LIN {X 0,Y 301.636,Z 553.215,A -85,B 0,C 180,E1 -16563.673,E2 -16563.673} C_VEL
LIN {X 0,Y 304.544,Z 543.643,A -85,B 0,C 180,E1 -16565.661,E2 -16565.661} C_VEL
LIN {X 0,Y 307.62,Z 532.508,A -85,B 0,C 180,E1 -16567.548,E2 -16567.548} C_VEL
LIN {X 0,Y 310.787,Z 520.04,A -85,B 0,C 180,E1 -16569.269,E2 -16569.269} C_VEL
LIN {X 0,Y 312.325,Z 513.549,A -85,B 0,C 180,E1 -16570.029,E2 -16570.029} C_VEL
LIN {X 0,Y 311.304,Z 507.375,A -85,B 0,C 180,E1 -16571.095,E2 -16571.095} C_VEL
LIN {X 0,Y 308.956,Z 499.343,A -85,B 0,C 180,E1 -16572.599,E2 -16572.599} C_VEL
LIN {X 0,Y 305.518,Z 490.599,A -85,B 0,C 180,E1 -16574.386,E2 -16574.386} C_VEL
LIN {X 0,Y 301.49,Z 482.379,A -85,B 0,C 180,E1 -16576.244,E2 -16576.244} C_VEL
LIN {X 0,Y 299.043,Z 478.041,A -85,B 0,C 180,E1 -16577.361,E2 -16577.361} C_VEL
LIN {X 0,Y 296.682,Z 474.656,A -85,B 0,C 180,E1 -16578.369,E2 -16578.369} C_VEL
LIN {X 0,Y 295.976,Z 473.129,A -85,B 0,C 180,E1 -16578.748,E2 -16578.748} C_VEL
LIN {X 0,Y 293.748,Z 470.591,A -85,B 0,C 180,E1 -16579.696,E2 -16579.696} C_VEL
LIN {X 0,Y 292.906,Z 468.275,A -85,B 0,C 180,E1 -16580.21,E2 -16580.21} C_VEL
LIN {X 0,Y 293.027,Z 467.949,A -85,B 0,C 180,E1 -16584.303,E2 -16584.303} C_VEL
LIN {X 0,Y 293.139,Z 468.076,A -85,B 0,C 180,E1 -16587.494,E2 -16587.494} C_VEL
LIN {X 0,Y 293.233,Z 468.47,A -85,B 0,C 180,E1 -16590.367,E2 -16590.367} C_VEL
LIN {X 0,Y 293.482,Z 469.78,A -85,B 0,C 180,E1 -16595.08,E2 -16595.08} C_VEL
LIN {X 0,Y 293.714,Z 471.269,A -85,B 0,C 180,E1 -16598.472,E2 -16598.472} C_VEL
LIN {X 0,Y 294.132,Z 473.425,A -85,B 0,C 180,E1 -16602.209,E2 -16602.209} C_VEL
LIN {X 0,Y 294.599,Z 476.404,A -85,B 0,C 180,E1 -16606.226,E2 -16606.226} C_VEL
LIN {X 0,Y 294.714,Z 478.064,A -85,B 0,C 180,E1 -16608.11,E2 -16608.11} C_VEL
LIN {X 0,Y 294.685,Z 479.821,A -85,B 0,C 180,E1 -16609.916,E2 -16609.916} C_VEL
LIN {X 0,Y 294.321,Z 482.209,A -85,B 0,C 180,E1 -16612.14,E2 -16612.14} C_VEL
LIN {X 0,Y 295.331,Z 485.828,A -85,B 0,C 180,E1 -16612.78,E2 -16612.78} C_VEL
LIN {X 0,Y 296.885,Z 488.688,A -85,B 0,C 180,E1 -16613.453,E2 -16613.453} C_VEL
LIN {X 0,Y 298.233,Z 492.616,A -85,B 0,C 180,E1 -16614.157,E2 -16614.157} C_VEL
LIN {X 0,Y 299.091,Z 494.768,A -85,B 0,C 180,E1 -16614.576,E2 -16614.576} C_VEL
LIN {X 0,Y 302.369,Z 504.747,A -85,B 0,C 180,E1 -16616.289,E2 -16616.289} C_VEL
LIN {X 0,Y 305.21,Z 516.489,A -85,B 0,C 180,E1 -16618.121,E2 -16618.121} C_VEL
LIN {X 0,Y 306.937,Z 528.969,A -85,B 0,C 180,E1 -16619.932,E2 -16619.932} C_VEL
LIN {X 0,Y 307.426,Z 538.705,A -85,B 0,C 180,E1 -16621.31,E2 -16621.31} C_VEL
LIN {X 0,Y 306.788,Z 549.97,A -85,B 0,C 180,E1 -16622.916,E2 -16622.916} C_VEL
LIN {X 0,Y 305.504,Z 555.839,A -85,B 0,C 180,E1 -16623.715,E2 -16623.715} C_VEL
LIN {X 0,Y 302.625,Z 566.34,A -85,B 0,C 180,E1 -16625.291,E2 -16625.291} C_VEL
LIN {X 0,Y 299.636,Z 576.972,A -85,B 0,C 180,E1 -16627.232,E2 -16627.232} C_VEL
LIN {X 0,Y 296.657,Z 587.405,A -85,B 0,C 180,E1 -16629.547,E2 -16629.547} C_VEL
LIN {X 0,Y 294.253,Z 596.056,A -85,B 0,C 180,E1 -16631.911,E2 -16631.911} C_VEL
LIN {X 0,Y 292.244,Z 604.121,A -85,B 0,C 180,E1 -16634.661,E2 -16634.661} C_VEL
LIN {X 0,Y 290.802,Z 610.467,A -85,B 0,C 180,E1 -16637.437,E2 -16637.437} C_VEL
LIN {X 0,Y 289.949,Z 615.257,A -85,B 0,C 180,E1 -16640.231,E2 -16640.231} C_VEL
LIN {X 0,Y 289.566,Z 618.621,A -85,B 0,C 180,E1 -16643.03,E2 -16643.03} C_VEL
LIN {X 0,Y 289.558,Z 620.61,A -85,B 0,C 180,E1 -16645.824,E2 -16645.824} C_VEL
LIN {X 0,Y 289.675,Z 621.212,A -85,B 0,C 180,E1 -16648.61,E2 -16648.61} C_VEL
LIN {X 0,Y 289.873,Z 620.996,A -85,B 0,C 180,E1 -16650,E2 -16650} C_VEL
LIN {X 0,Y 289.631,Z 619.447,A -85,B 0,C 180,E1 -16652.782,E2 -16652.782} C_VEL
LIN {X 0,Y 289.672,Z 618.137,A -85,B 0,C 180,E1 -16654.174,E2 -16654.174} C_VEL
LIN {X 0,Y 289.71,Z 615.903,A -85,B 0,C 180,E1 -16655.954,E2 -16655.954} C_VEL
LIN {X 0,Y 289.811,Z 611.833,A -85,B 0,C 180,E1 -16658.366,E2 -16658.366} C_VEL
LIN {X 0,Y 290.092,Z 607.241,A -85,B 0,C 180,E1 -16660.469,E2 -16660.469} C_VEL
LIN {X 0,Y 290.817,Z 600.58,A -85,B 0,C 180,E1 -16662.917,E2 -16662.917} C_VEL
LIN {X 0,Y 291.753,Z 592.22,A -85,B 0,C 180,E1 -16665.365,E2 -16665.365} C_VEL
LIN {X 0,Y 293.093,Z 583.538,A -85,B 0,C 180,E1 -16667.441,E2 -16667.441} C_VEL
LIN {X 0,Y 294.652,Z 573.049,A -85,B 0,C 180,E1 -16669.507,E2 -16669.507} C_VEL
LIN {X 0,Y 296.588,Z 561.479,A -85,B 0,C 180,E1 -16671.366,E2 -16671.366} C_VEL
LIN {X 0,Y 298.446,Z 548.652,A -85,B 0,C 180,E1 -16673.047,E2 -16673.047} C_VEL
LIN {X 0,Y 298.999,Z 544.142,A -85,B 0,C 180,E1 -16673.552,E2 -16673.552} C_VEL
LIN {X 0,Y 297.569,Z 530.241,A -85,B 0,C 180,E1 -16675.065,E2 -16675.065} C_VEL
LIN {X 0,Y 295.6,Z 515.743,A -85,B 0,C 180,E1 -16676.36,E2 -16676.36} C_VEL
LIN {X 0,Y 293.096,Z 500.193,A -85,B 0,C 180,E1 -16677.476,E2 -16677.476} C_VEL
LIN {X 0,Y 291.412,Z 490.807,A -85,B 0,C 180,E1 -16678.051,E2 -16678.051} C_VEL
LIN {X 0,Y 292.233,Z 484.923,A -85,B 0,C 180,E1 -16681.943,E2 -16681.943} C_VEL
LIN {X 0,Y 293.22,Z 478.9,A -85,B 0,C 180,E1 -16686.02,E2 -16686.02} C_VEL
LIN {X 0,Y 293.911,Z 474.253,A -85,B 0,C 180,E1 -16689.252,E2 -16689.252} C_VEL
LIN {X 0,Y 293.611,Z 470.39,A -85,B 0,C 180,E1 -16692.096,E2 -16692.096} C_VEL
LIN {X 0,Y 292.747,Z 465.551,A -85,B 0,C 180,E1 -16695.877,E2 -16695.877} C_VEL
LIN {X 0,Y 291.997,Z 461.184,A -85,B 0,C 180,E1 -16699.469,E2 -16699.469} C_VEL
LIN {X 0,Y 291.434,Z 457.811,A -85,B 0,C 180,E1 -16702.434,E2 -16702.434} C_VEL
LIN {X 0,Y 291.342,Z 457.816,A -85,B 0,C 180,E1 -16706.301,E2 -16706.301} C_VEL
LIN {X 0,Y 291.384,Z 457.812,A -85,B 0,C 180,E1 -16710.259,E2 -16710.259} C_VEL
LIN {X 0,Y 291.412,Z 457.807,A -85,B 0,C 180,E1 -16714.272,E2 -16714.272} C_VEL
LIN {X 0,Y 291.377,Z 457.814,A -85,B 0,C 180,E1 -16717.299,E2 -16717.299} C_VEL
LIN {X 0,Y 291.454,Z 457.803,A -85,B 0,C 180,E1 -16720.27,E2 -16720.27} C_VEL
LIN {X 0,Y 291.551,Z 457.793,A -85,B 0,C 180,E1 -16724.624,E2 -16724.624} C_VEL
LIN {X 0,Y 291.532,Z 457.797,A -85,B 0,C 180,E1 -16728.881,E2 -16728.881} C_VEL
LIN {X 0,Y 291.704,Z 457.771,A -85,B 0,C 180,E1 -16731.689,E2 -16731.689} C_VEL
LIN {X 0,Y 291.627,Z 457.783,A -85,B 0,C 180,E1 -16734.469,E2 -16734.469} C_VEL
LIN {X 0,Y 291.886,Z 457.754,A -85,B 0,C 180,E1 -16738.621,E2 -16738.621} C_VEL
LIN {X 0,Y 291.888,Z 457.748,A -85,B 0,C 180,E1 -16741.38,E2 -16741.38} C_VEL
LIN {X 0,Y 291.744,Z 457.768,A -85,B 0,C 180,E1 -16746.918,E2 -16746.918} C_VEL
LIN {X 0,Y 291.625,Z 457.781,A -85,B 0,C 180,E1 -16749.712,E2 -16749.712} C_VEL
LIN {X 0,Y 291.517,Z 457.796,A -85,B 0,C 180,E1 -16753.951,E2 -16753.951} C_VEL
LIN {X 0,Y 291.483,Z 457.8,A -85,B 0,C 180,E1 -16756.818,E2 -16756.818} C_VEL
LIN {X 0,Y 291.447,Z 457.804,A -85,B 0,C 180,E1 -16759.875,E2 -16759.875} C_VEL
LIN {X 0,Y 291.397,Z 457.814,A -85,B 0,C 180,E1 -16764.206,E2 -16764.206} C_VEL
LIN {X 0,Y 291.419,Z 457.806,A -85,B 0,C 180,E1 -16767.272,E2 -16767.272} C_VEL
LIN {X 0,Y 291.334,Z 457.82,A -85,B 0,C 180,E1 -16770.438,E2 -16770.438} C_VEL
LIN {X 0,Y 291.342,Z 457.818,A -85,B 0,C 180,E1 -16773.699,E2 -16773.699} C_VEL
LIN {X 0,Y 291.379,Z 457.811,A -85,B 0,C 180,E1 -16777.256,E2 -16777.256} C_VEL
LIN {X 0,Y 291.332,Z 457.819,A -85,B 0,C 180,E1 -16780.643,E2 -16780.643} C_VEL
LIN {X 0,Y 291.289,Z 457.824,A -85,B 0,C 180,E1 -16784.403,E2 -16784.403} C_VEL
LIN {X 0,Y 291.355,Z 457.816,A -85,B 0,C 180,E1 -16788.399,E2 -16788.399} C_VEL
LIN {X 0,Y 291.38,Z 457.812,A -85,B 0,C 180,E1 -16791.163,E2 -16791.163} C_VEL
LIN {X 0,Y 291.386,Z 457.81,A -85,B 0,C 180,E1 -16794.63,E2 -16794.63} C_VEL
LIN {X 0,Y 291.374,Z 457.816,A -85,B 0,C 180,E1 -16797.952,E2 -16797.952} C_VEL
LIN {X 0,Y 291.391,Z 457.811,A -85,B 0,C 180,E1 -16801.16,E2 -16801.16} C_VEL
LIN {X 0,Y 291.423,Z 457.807,A -85,B 0,C 180,E1 -16804.273,E2 -16804.273} C_VEL
LIN {X 0,Y 291.384,Z 457.813,A -85,B 0,C 180,E1 -16807.3,E2 -16807.3} C_VEL
LIN {X 0,Y 291.461,Z 457.802,A -85,B 0,C 180,E1 -16810.271,E2 -16810.271} C_VEL
LIN {X 0,Y 291.558,Z 457.789,A -85,B 0,C 180,E1 -16814.624,E2 -16814.624} C_VEL
LIN {X 0,Y 291.539,Z 457.792,A -85,B 0,C 180,E1 -16818.881,E2 -16818.881} C_VEL
LIN {X 0,Y 291.658,Z 457.78,A -85,B 0,C 180,E1 -16821.687,E2 -16821.687} C_VEL
LIN {X 0,Y 291.615,Z 457.782,A -85,B 0,C 180,E1 -16824.468,E2 -16824.468} C_VEL
LIN {X 0,Y 291.892,Z 457.747,A -85,B 0,C 180,E1 -16828.62,E2 -16828.62} C_VEL
LIN {X 0,Y 291.892,Z 457.752,A -85,B 0,C 180,E1 -16831.38,E2 -16831.38} C_VEL
LIN {X 0,Y 291.738,Z 457.769,A -85,B 0,C 180,E1 -16836.918,E2 -16836.918} C_VEL
LIN {X 0,Y 291.578,Z 457.787,A -85,B 0,C 180,E1 -16839.713,E2 -16839.713} C_VEL
LIN {X 0,Y 291.525,Z 457.794,A -85,B 0,C 180,E1 -16843.95,E2 -16843.95} C_VEL
LIN {X 0,Y 291.49,Z 457.8,A -85,B 0,C 180,E1 -16846.817,E2 -16846.817} C_VEL
LIN {X 0,Y 291.453,Z 457.803,A -85,B 0,C 180,E1 -16849.874,E2 -16849.874} C_VEL
LIN {X 0,Y 291.402,Z 457.809,A -85,B 0,C 180,E1 -16854.205,E2 -16854.205} C_VEL
LIN {X 0,Y 291.424,Z 457.81,A -85,B 0,C 180,E1 -16857.271,E2 -16857.271} C_VEL
LIN {X 0,Y 291.336,Z 457.819,A -85,B 0,C 180,E1 -16860.436,E2 -16860.436} C_VEL
LIN {X 0,Y 291.243,Z 457.829,A -85,B 0,C 180,E1 -16863.711,E2 -16863.711} C_VEL
LIN {X 0,Y 290.986,Z 457.864,A -85,B 0,C 180,E1 -16867.152,E2 -16867.152} C_VEL
LIN {X 0,Y 290.57,Z 457.917,A -85,B 0,C 180,E1 -16870.771,E2 -16870.771} C_VEL
LIN {X 0,Y 290.267,Z 458.188,A -85,B 0,C 180,E1 -16873.417,E2 -16873.417} C_VEL
LIN {X 0,Y 290.253,Z 458.716,A -85,B 0,C 180,E1 -16874.108,E2 -16874.108} C_VEL
LIN {X 0,Y 295.016,Z 475.364,A -85,B 0,C 180,E1 -16875.334,E2 -16875.334} C_VEL
LIN {X 0,Y 298.444,Z 488.673,A -85,B 0,C 180,E1 -16876.532,E2 -16876.532} C_VEL
LIN {X 0,Y 300.997,Z 500.048,A -85,B 0,C 180,E1 -16877.735,E2 -16877.735} C_VEL
LIN {X 0,Y 299.772,Z 511.987,A -85,B 0,C 180,E1 -16878.97,E2 -16878.97} C_VEL
LIN {X 0,Y 298.086,Z 523.963,A -85,B 0,C 180,E1 -16880.462,E2 -16880.462} C_VEL
LIN {X 0,Y 296.452,Z 535.158,A -85,B 0,C 180,E1 -16882.162,E2 -16882.162} C_VEL
LIN {X 0,Y 294.809,Z 545.907,A -85,B 0,C 180,E1 -16884.146,E2 -16884.146} C_VEL
LIN {X 0,Y 293.434,Z 554.954,A -85,B 0,C 180,E1 -16886.161,E2 -16886.161} C_VEL
LIN {X 0,Y 292.141,Z 563.427,A -85,B 0,C 180,E1 -16888.45,E2 -16888.45} C_VEL
LIN {X 0,Y 291.228,Z 570.208,A -85,B 0,C 180,E1 -16890.689,E2 -16890.689} C_VEL
LIN {X 0,Y 290.465,Z 576.263,A -85,B 0,C 180,E1 -16893.175,E2 -16893.175} C_VEL
LIN {X 0,Y 289.946,Z 580.967,A -85,B 0,C 180,E1 -16895.665,E2 -16895.665} C_VEL
LIN {X 0,Y 289.734,Z 583.225,A -85,B 0,C 180,E1 -16897.181,E2 -16897.181} C_VEL
LIN {X 0,Y 289.45,Z 586.399,A -85,B 0,C 180,E1 -16900.127,E2 -16900.127} C_VEL
LIN {X 0,Y 289.497,Z 587.383,A -85,B 0,C 180,E1 -16901.603,E2 -16901.603} C_VEL
LIN {X 0,Y 289.655,Z 588.2,A -85,B 0,C 180,E1 -16904.52,E2 -16904.52} C_VEL
LIN {X 0,Y 290.106,Z 587.576,A -85,B 0,C 180,E1 -16907.406,E2 -16907.406} C_VEL
LIN {X 0,Y 290.896,Z 585.558,A -85,B 0,C 180,E1 -16910.263,E2 -16910.263} C_VEL
LIN {X 0,Y 292.112,Z 582.127,A -85,B 0,C 180,E1 -16913.09,E2 -16913.09} C_VEL
LIN {X 0,Y 293.789,Z 577.212,A -85,B 0,C 180,E1 -16915.884,E2 -16915.884} C_VEL
LIN {X 0,Y 296.006,Z 570.651,A -85,B 0,C 180,E1 -16918.639,E2 -16918.639} C_VEL
LIN {X 0,Y 296.133,Z 570.261,A -85,B 0,C 180,E1 -16918.78,E2 -16918.78} C_VEL
LIN {X 0,Y 296.44,Z 567.593,A -85,B 0,C 180,E1 -16919.797,E2 -16919.797} C_VEL
LIN {X 0,Y 295.401,Z 563.24,A -85,B 0,C 180,E1 -16921.513,E2 -16921.513} C_VEL
LIN {X 0,Y 294.562,Z 558.444,A -85,B 0,C 180,E1 -16923.185,E2 -16923.185} C_VEL
LIN {X 0,Y 295.151,Z 555.046,A -85,B 0,C 180,E1 -16924.112,E2 -16924.112} C_VEL
LIN {X 0,Y 298.125,Z 545.908,A -85,B 0,C 180,E1 -16926.105,E2 -16926.105} C_VEL
LIN {X 0,Y 301.368,Z 535.215,A -85,B 0,C 180,E1 -16928.043,E2 -16928.043} C_VEL
LIN {X 0,Y 304.666,Z 523.197,A -85,B 0,C 180,E1 -16929.795,E2 -16929.795} C_VEL
LIN {X 0,Y 306.496,Z 515.55,A -85,B 0,C 180,E1 -16930.745,E2 -16930.745} C_VEL
LIN {X 0,Y 305.179,Z 508.082,A -85,B 0,C 180,E1 -16932.161,E2 -16932.161} C_VEL
LIN {X 0,Y 302.061,Z 498.218,A -85,B 0,C 180,E1 -16934.202,E2 -16934.202} C_VEL
LIN {X 0,Y 297.217,Z 487.393,A -85,B 0,C 180,E1 -16936.79,E2 -16936.79} C_VEL
LIN {X 0,Y 294.604,Z 482.84,A -85,B 0,C 180,E1 -16938.067,E2 -16938.067} C_VEL
LIN {X 0,Y 291.609,Z 478.107,A -85,B 0,C 180,E1 -16939.582,E2 -16939.582} C_VEL
LIN {X 0,Y 289.874,Z 475.066,A -85,B 0,C 180,E1 -16940.55,E2 -16940.55} C_VEL
LIN {X 0,Y 289.424,Z 474.387,A -85,B 0,C 180,E1 -16940.797,E2 -16940.797} C_VEL
LIN {X 0,Y 287.052,Z 472.053,A -85,B 0,C 180,E1 -16941.97,E2 -16941.97} C_VEL
LIN {X 0,Y 286.042,Z 469.515,A -85,B 0,C 180,E1 -16942.728,E2 -16942.728} C_VEL
LIN {X 0,Y 286.142,Z 469.511,A -85,B 0,C 180,E1 -16946.238,E2 -16946.238} C_VEL
LIN {X 0,Y 286.237,Z 469.877,A -85,B 0,C 180,E1 -16949.41,E2 -16949.41} C_VEL
LIN {X 0,Y 286.413,Z 470.819,A -85,B 0,C 180,E1 -16953.459,E2 -16953.459} C_VEL
LIN {X 0,Y 286.746,Z 472.49,A -85,B 0,C 180,E1 -16957.787,E2 -16957.787} C_VEL
LIN {X 0,Y 287.094,Z 474.43,A -85,B 0,C 180,E1 -16961.373,E2 -16961.373} C_VEL
LIN {X 0,Y 287.528,Z 477.024,A -85,B 0,C 180,E1 -16965.141,E2 -16965.141} C_VEL
LIN {X 0,Y 287.714,Z 478.619,A -85,B 0,C 180,E1 -16967.122,E2 -16967.122} C_VEL
LIN {X 0,Y 287.741,Z 481.304,A -85,B 0,C 180,E1 -16969.887,E2 -16969.887} C_VEL
LIN {X 0,Y 288.623,Z 484.501,A -85,B 0,C 180,E1 -16970.542,E2 -16970.542} C_VEL
LIN {X 0,Y 290.726,Z 488.229,A -85,B 0,C 180,E1 -16971.611,E2 -16971.611} C_VEL
LIN {X 0,Y 292.274,Z 492.398,A -85,B 0,C 180,E1 -16972.515,E2 -16972.515} C_VEL
LIN {X 0,Y 293.032,Z 494.501,A -85,B 0,C 180,E1 -16972.961,E2 -16972.961} C_VEL
LIN {X 0,Y 295.012,Z 500.212,A -85,B 0,C 180,E1 -16974.093,E2 -16974.093} C_VEL
LIN {X 0,Y 297.161,Z 507.283,A -85,B 0,C 180,E1 -16975.417,E2 -16975.417} C_VEL
LIN {X 0,Y 299.741,Z 518.981,A -85,B 0,C 180,E1 -16977.366,E2 -16977.366} C_VEL
LIN {X 0,Y 301.182,Z 530.305,A -85,B 0,C 180,E1 -16979.112,E2 -16979.112} C_VEL
LIN {X 0,Y 301.471,Z 540.725,A -85,B 0,C 180,E1 -16980.689,E2 -16980.689} C_VEL
LIN {X 0,Y 300.65,Z 551.565,A -85,B 0,C 180,E1 -16982.316,E2 -16982.316} C_VEL
LIN {X 0,Y 298.932,Z 558.293,A -85,B 0,C 180,E1 -16983.28,E2 -16983.28} C_VEL
LIN {X 0,Y 295.705,Z 569.214,A -85,B 0,C 180,E1 -16985.048,E2 -16985.048} C_VEL
LIN {X 0,Y 292.682,Z 579.34,A -85,B 0,C 180,E1 -16987.033,E2 -16987.033} C_VEL
LIN {X 0,Y 289.615,Z 589.228,A -85,B 0,C 180,E1 -16989.399,E2 -16989.399} C_VEL
LIN {X 0,Y 287.19,Z 597.442,A -85,B 0,C 180,E1 -16991.82,E2 -16991.82} C_VEL
LIN {X 0,Y 285.366,Z 604.23,A -85,B 0,C 180,E1 -16994.282,E2 -16994.282} C_VEL
LIN {X 0,Y 283.848,Z 610.397,A -85,B 0,C 180,E1 -16997.124,E2 -16997.124} C_VEL
LIN {X 0,Y 282.886,Z 615.084,A -85,B 0,C 180,E1 -16999.985,E2 -16999.985} C_VEL
LIN {X 0,Y 282.484,Z 618.345,A -85,B 0,C 180,E1 -17002.854,E2 -17002.854} C_VEL
LIN {X 0,Y 282.472,Z 620.237,A -85,B 0,C 180,E1 -17005.719,E2 -17005.719} C_VEL
LIN {X 0,Y 282.584,Z 620.751,A -85,B 0,C 180,E1 -17008.575,E2 -17008.575} C_VEL
LIN {X 0,Y 282.801,Z 620.49,A -85,B 0,C 180,E1 -17010,E2 -17010} C_VEL
LIN {X 0,Y 282.555,Z 618.847,A -85,B 0,C 180,E1 -17012.851,E2 -17012.851} C_VEL
LIN {X 0,Y 282.61,Z 617.487,A -85,B 0,C 180,E1 -17014.278,E2 -17014.278} C_VEL
LIN {X 0,Y 282.646,Z 615.367,A -85,B 0,C 180,E1 -17015.957,E2 -17015.957} C_VEL
LIN {X 0,Y 282.744,Z 610.982,A -85,B 0,C 180,E1 -17018.577,E2 -17018.577} C_VEL
LIN {X 0,Y 283.058,Z 606.337,A -85,B 0,C 180,E1 -17020.732,E2 -17020.732} C_VEL
LIN {X 0,Y 283.824,Z 599.54,A -85,B 0,C 180,E1 -17023.241,E2 -17023.241} C_VEL
LIN {X 0,Y 284.87,Z 591.046,A -85,B 0,C 180,E1 -17025.746,E2 -17025.746} C_VEL
LIN {X 0,Y 286.245,Z 582.229,A -85,B 0,C 180,E1 -17027.872,E2 -17027.872} C_VEL
LIN {X 0,Y 287.88,Z 571.595,A -85,B 0,C 180,E1 -17029.985,E2 -17029.985} C_VEL
LIN {X 0,Y 289.861,Z 559.834,A -85,B 0,C 180,E1 -17031.887,E2 -17031.887} C_VEL
LIN {X 0,Y 291.651,Z 547.852,A -85,B 0,C 180,E1 -17033.467,E2 -17033.467} C_VEL
LIN {X 0,Y 292.019,Z 544.439,A -85,B 0,C 180,E1 -17033.859,E2 -17033.859} C_VEL
LIN {X 0,Y 290.737,Z 531.607,A -85,B 0,C 180,E1 -17035.312,E2 -17035.312} C_VEL
LIN {X 0,Y 288.918,Z 517.699,A -85,B 0,C 180,E1 -17036.627,E2 -17036.627} C_VEL
LIN {X 0,Y 286.552,Z 502.648,A -85,B 0,C 180,E1 -17037.774,E2 -17037.774} C_VEL
LIN {X 0,Y 284.415,Z 490.492,A -85,B 0,C 180,E1 -17038.536,E2 -17038.536} C_VEL
LIN {X 0,Y 285.176,Z 485.419,A -85,B 0,C 180,E1 -17041.995,E2 -17041.995} C_VEL
LIN {X 0,Y 286.177,Z 479.481,A -85,B 0,C 180,E1 -17046.114,E2 -17046.114} C_VEL
LIN {X 0,Y 286.862,Z 474.662,A -85,B 0,C 180,E1 -17049.567,E2 -17049.567} C_VEL
LIN {X 0,Y 286.483,Z 470.667,A -85,B 0,C 180,E1 -17052.612,E2 -17052.612} C_VEL
LIN {X 0,Y 285.616,Z 465.894,A -85,B 0,C 180,E1 -17056.451,E2 -17056.451} C_VEL
LIN {X 0,Y 284.848,Z 461.598,A -85,B 0,C 180,E1 -17060.097,E2 -17060.097} C_VEL
LIN {X 0,Y 284.412,Z 458.685,A -85,B 0,C 180,E1 -17062.746,E2 -17062.746} C_VEL
LIN {X 0,Y 284.303,Z 458.698,A -85,B 0,C 180,E1 -17067.055,E2 -17067.055} C_VEL
LIN {X 0,Y 284.356,Z 458.688,A -85,B 0,C 180,E1 -17070.376,E2 -17070.376} C_VEL
LIN {X 0,Y 284.374,Z 458.684,A -85,B 0,C 180,E1 -17073.586,E2 -17073.586} C_VEL
LIN {X 0,Y 284.362,Z 458.688,A -85,B 0,C 180,E1 -17076.707,E2 -17076.707} C_VEL
LIN {X 0,Y 284.399,Z 458.683,A -85,B 0,C 180,E1 -17081.262,E2 -17081.262} C_VEL
LIN {X 0,Y 284.488,Z 458.671,A -85,B 0,C 180,E1 -17084.459,E2 -17084.459} C_VEL
LIN {X 0,Y 284.484,Z 458.674,A -85,B 0,C 180,E1 -17088.602,E2 -17088.602} C_VEL
LIN {X 0,Y 284.654,Z 458.649,A -85,B 0,C 180,E1 -17091.481,E2 -17091.481} C_VEL
LIN {X 0,Y 284.597,Z 458.658,A -85,B 0,C 180,E1 -17094.331,E2 -17094.331} C_VEL
LIN {X 0,Y 284.852,Z 458.63,A -85,B 0,C 180,E1 -17098.587,E2 -17098.587} C_VEL
LIN {X 0,Y 284.854,Z 458.623,A -85,B 0,C 180,E1 -17101.414,E2 -17101.414} C_VEL
LIN {X 0,Y 284.695,Z 458.645,A -85,B 0,C 180,E1 -17107.09,E2 -17107.09} C_VEL
LIN {X 0,Y 284.562,Z 458.661,A -85,B 0,C 180,E1 -17109.956,E2 -17109.956} C_VEL
LIN {X 0,Y 284.474,Z 458.676,A -85,B 0,C 180,E1 -17114.304,E2 -17114.304} C_VEL
LIN {X 0,Y 284.421,Z 458.678,A -85,B 0,C 180,E1 -17117.249,E2 -17117.249} C_VEL
LIN {X 0,Y 284.375,Z 458.687,A -85,B 0,C 180,E1 -17120.243,E2 -17120.243} C_VEL
LIN {X 0,Y 284.366,Z 458.687,A -85,B 0,C 180,E1 -17123.876,E2 -17123.876} C_VEL
LIN {X 0,Y 284.394,Z 458.681,A -85,B 0,C 180,E1 -17127.174,E2 -17127.174} C_VEL
LIN {X 0,Y 284.293,Z 458.694,A -85,B 0,C 180,E1 -17131.275,E2 -17131.275} C_VEL
LIN {X 0,Y 284.339,Z 458.689,A -85,B 0,C 180,E1 -17135.349,E2 -17135.349} C_VEL
LIN {X 0,Y 284.317,Z 458.696,A -85,B 0,C 180,E1 -17138.169,E2 -17138.169} C_VEL
LIN {X 0,Y 284.268,Z 458.702,A -85,B 0,C 180,E1 -17142.125,E2 -17142.125} C_VEL
LIN {X 0,Y 284.272,Z 458.7,A -85,B 0,C 180,E1 -17146.193,E2 -17146.193} C_VEL
LIN {X 0,Y 284.351,Z 458.692,A -85,B 0,C 180,E1 -17150.014,E2 -17150.014} C_VEL
LIN {X 0,Y 284.353,Z 458.689,A -85,B 0,C 180,E1 -17153.618,E2 -17153.618} C_VEL
LIN {X 0,Y 284.309,Z 458.693,A -85,B 0,C 180,E1 -17157.19,E2 -17157.19} C_VEL
LIN {X 0,Y 284.363,Z 458.686,A -85,B 0,C 180,E1 -17160.377,E2 -17160.377} C_VEL
LIN {X 0,Y 284.383,Z 458.686,A -85,B 0,C 180,E1 -17163.588,E2 -17163.588} C_VEL
LIN {X 0,Y 284.369,Z 458.685,A -85,B 0,C 180,E1 -17166.708,E2 -17166.708} C_VEL
LIN {X 0,Y 284.407,Z 458.682,A -85,B 0,C 180,E1 -17171.262,E2 -17171.262} C_VEL
LIN {X 0,Y 284.495,Z 458.669,A -85,B 0,C 180,E1 -17174.459,E2 -17174.459} C_VEL
LIN {X 0,Y 284.491,Z 458.67,A -85,B 0,C 180,E1 -17178.602,E2 -17178.602} C_VEL
LIN {X 0,Y 284.615,Z 458.658,A -85,B 0,C 180,E1 -17181.48,E2 -17181.48} C_VEL
LIN {X 0,Y 284.583,Z 458.658,A -85,B 0,C 180,E1 -17184.331,E2 -17184.331} C_VEL
LIN {X 0,Y 284.858,Z 458.624,A -85,B 0,C 180,E1 -17188.586,E2 -17188.586} C_VEL
LIN {X 0,Y 284.858,Z 458.629,A -85,B 0,C 180,E1 -17191.414,E2 -17191.414} C_VEL
LIN {X 0,Y 284.689,Z 458.648,A -85,B 0,C 180,E1 -17197.09,E2 -17197.09} C_VEL
LIN {X 0,Y 284.522,Z 458.665,A -85,B 0,C 180,E1 -17199.957,E2 -17199.957} C_VEL
LIN {X 0,Y 284.485,Z 458.671,A -85,B 0,C 180,E1 -17204.302,E2 -17204.302} C_VEL
LIN {X 0,Y 284.428,Z 458.681,A -85,B 0,C 180,E1 -17207.248,E2 -17207.248} C_VEL
LIN {X 0,Y 284.381,Z 458.684,A -85,B 0,C 180,E1 -17210.242,E2 -17210.242} C_VEL
LIN {X 0,Y 284.371,Z 458.685,A -85,B 0,C 180,E1 -17213.875,E2 -17213.875} C_VEL
LIN {X 0,Y 284.399,Z 458.686,A -85,B 0,C 180,E1 -17217.173,E2 -17217.173} C_VEL
LIN {X 0,Y 284.315,Z 458.692,A -85,B 0,C 180,E1 -17220.097,E2 -17220.097} C_VEL
LIN {X 0,Y 284.236,Z 458.707,A -85,B 0,C 180,E1 -17222.954,E2 -17222.954} C_VEL
LIN {X 0,Y 283.992,Z 458.734,A -85,B 0,C 180,E1 -17226.436,E2 -17226.436} C_VEL
LIN {X 0,Y 283.581,Z 458.789,A -85,B 0,C 180,E1 -17230.117,E2 -17230.117} C_VEL
LIN {X 0,Y 283.212,Z 459.066,A -85,B 0,C 180,E1 -17233.562,E2 -17233.562} C_VEL
LIN {X 0,Y 288.337,Z 477.065,A -85,B 0,C 180,E1 -17234.978,E2 -17234.978} C_VEL
LIN {X 0,Y 292.069,Z 492.048,A -85,B 0,C 180,E1 -17236.409,E2 -17236.409} C_VEL
LIN {X 0,Y 294.193,Z 501.757,A -85,B 0,C 180,E1 -17237.474,E2 -17237.474} C_VEL
LIN {X 0,Y 292.589,Z 514.732,A -85,B 0,C 180,E1 -17238.886,E2 -17238.886} C_VEL
LIN {X 0,Y 290.876,Z 526.774,A -85,B 0,C 180,E1 -17240.496,E2 -17240.496} C_VEL
LIN {X 0,Y 289.116,Z 538.212,A -85,B 0,C 180,E1 -17242.355,E2 -17242.355} C_VEL
LIN {X 0,Y 287.453,Z 549.046,A -85,B 0,C 180,E1 -17244.502,E2 -17244.502} C_VEL
LIN {X 0,Y 285.955,Z 558.102,A -85,B 0,C 180,E1 -17246.68,E2 -17246.68} C_VEL
LIN {X 0,Y 284.869,Z 565.363,A -85,B 0,C 180,E1 -17248.795,E2 -17248.795} C_VEL
LIN {X 0,Y 284.001,Z 572.022,A -85,B 0,C 180,E1 -17251.147,E2 -17251.147} C_VEL
LIN {X 0,Y 283.303,Z 577.349,A -85,B 0,C 180,E1 -17253.478,E2 -17253.478} C_VEL
LIN {X 0,Y 282.83,Z 581.53,A -85,B 0,C 180,E1 -17255.794,E2 -17255.794} C_VEL
LIN {X 0,Y 282.51,Z 584.684,A -85,B 0,C 180,E1 -17258.089,E2 -17258.089} C_VEL
LIN {X 0,Y 282.377,Z 587.411,A -85,B 0,C 180,E1 -17261.122,E2 -17261.122} C_VEL
LIN {X 0,Y 282.509,Z 588.606,A -85,B 0,C 180,E1 -17264.118,E2 -17264.118} C_VEL
LIN {X 0,Y 282.77,Z 588.648,A -85,B 0,C 180,E1 -17265.764,E2 -17265.764} C_VEL
LIN {X 0,Y 283.309,Z 587.683,A -85,B 0,C 180,E1 -17268.553,E2 -17268.553} C_VEL
LIN {X 0,Y 284.328,Z 585.272,A -85,B 0,C 180,E1 -17271.471,E2 -17271.471} C_VEL
LIN {X 0,Y 285.727,Z 581.476,A -85,B 0,C 180,E1 -17274.353,E2 -17274.353} C_VEL
LIN {X 0,Y 287.71,Z 576.164,A -85,B 0,C 180,E1 -17277.199,E2 -17277.199} C_VEL
LIN {X 0,Y 290.217,Z 569.214,A -85,B 0,C 180,E1 -17280,E2 -17280} C_VEL
LIN {X 0,Y 292.878,Z 561.626,A -85,B 0,C 180,E1 -17282.406,E2 -17282.406} C_VEL
LIN {X 0,Y 295.151,Z 555.046,A -85,B 0,C 180,E1 -17284.112,E2 -17284.112} C_VEL
LIN {X 0,Y 295.819,Z 551.514,A -85,B 0,C 180,E1 -17285.023,E2 -17285.023} C_VEL
LIN {X 0,Y 295.424,Z 545.885,A -85,B 0,C 180,E1 -17286.606,E2 -17286.606} C_VEL
LIN {X 0,Y 295.099,Z 539.845,A -85,B 0,C 180,E1 -17288.125,E2 -17288.125} C_VEL
LIN {X 0,Y 295.833,Z 535.677,A -85,B 0,C 180,E1 -17288.919,E2 -17288.919} C_VEL
LIN {X 0,Y 299.596,Z 522.778,A -85,B 0,C 180,E1 -17290.816,E2 -17290.816} C_VEL
LIN {X 0,Y 300.846,Z 517.861,A -85,B 0,C 180,E1 -17291.453,E2 -17291.453} C_VEL
LIN {X 0,Y 299.148,Z 509.188,A -85,B 0,C 180,E1 -17293.243,E2 -17293.243} C_VEL
LIN {X 0,Y 296.526,Z 500.962,A -85,B 0,C 180,E1 -17295.112,E2 -17295.112} C_VEL
LIN {X 0,Y 292.746,Z 492.122,A -85,B 0,C 180,E1 -17297.409,E2 -17297.409} C_VEL
LIN {X 0,Y 289.042,Z 485.159,A -85,B 0,C 180,E1 -17299.532,E2 -17299.532} C_VEL
LIN {X 0,Y 286.075,Z 480.427,A -85,B 0,C 180,E1 -17301.28,E2 -17301.28} C_VEL
LIN {X 0,Y 284.028,Z 477.985,A -85,B 0,C 180,E1 -17302.457,E2 -17302.457} C_VEL
LIN {X 0,Y 283.006,Z 475.883,A -85,B 0,C 180,E1 -17303.246,E2 -17303.246} C_VEL
LIN {X 0,Y 280.604,Z 473.931,A -85,B 0,C 180,E1 -17304.723,E2 -17304.723} C_VEL
LIN {X 0,Y 279.324,Z 471.565,A -85,B 0,C 180,E1 -17305.863,E2 -17305.863} C_VEL
LIN {X 0,Y 279.211,Z 471.04,A -85,B 0,C 180,E1 -17306.055,E2 -17306.055} C_VEL
LIN {X 0,Y 279.348,Z 471.577,A -85,B 0,C 180,E1 -17310.21,E2 -17310.21} C_VEL
LIN {X 0,Y 279.52,Z 472.549,A -85,B 0,C 180,E1 -17313.931,E2 -17313.931} C_VEL
LIN {X 0,Y 279.727,Z 473.749,A -85,B 0,C 180,E1 -17317.084,E2 -17317.084} C_VEL
LIN {X 0,Y 280.16,Z 475.855,A -85,B 0,C 180,E1 -17321.188,E2 -17321.188} C_VEL
LIN {X 0,Y 280.516,Z 478.051,A -85,B 0,C 180,E1 -17324.548,E2 -17324.548} C_VEL
LIN {X 0,Y 280.758,Z 479.871,A -85,B 0,C 180,E1 -17326.788,E2 -17326.788} C_VEL
LIN {X 0,Y 281.991,Z 483.552,A -85,B 0,C 180,E1 -17327.833,E2 -17327.833} C_VEL
LIN {X 0,Y 284.415,Z 487.266,A -85,B 0,C 180,E1 -17329.308,E2 -17329.308} C_VEL
LIN {X 0,Y 285.878,Z 491.396,A -85,B 0,C 180,E1 -17330.351,E2 -17330.351} C_VEL
LIN {X 0,Y 286.995,Z 493.604,A -85,B 0,C 180,E1 -17331.015,E2 -17331.015} C_VEL
LIN {X 0,Y 288.952,Z 499.288,A -85,B 0,C 180,E1 -17332.31,E2 -17332.31} C_VEL
LIN {X 0,Y 291.59,Z 507.954,A -85,B 0,C 180,E1 -17334.121,E2 -17334.121} C_VEL
LIN {X 0,Y 294.245,Z 520.824,A -85,B 0,C 180,E1 -17336.453,E2 -17336.453} C_VEL
LIN {X 0,Y 295.495,Z 532.839,A -85,B 0,C 180,E1 -17338.451,E2 -17338.451} C_VEL
LIN {X 0,Y 295.602,Z 542.862,A -85,B 0,C 180,E1 -17340.048,E2 -17340.048} C_VEL
LIN {X 0,Y 294.535,Z 553.318,A -85,B 0,C 180,E1 -17341.71,E2 -17341.71} C_VEL
LIN {X 0,Y 291.13,Z 564.74,A -85,B 0,C 180,E1 -17343.469,E2 -17343.469} C_VEL
LIN {X 0,Y 287.663,Z 575.387,A -85,B 0,C 180,E1 -17345.46,E2 -17345.46} C_VEL
LIN {X 0,Y 284.318,Z 585.794,A -85,B 0,C 180,E1 -17347.855,E2 -17347.855} C_VEL
LIN {X 0,Y 281.493,Z 594.475,A -85,B 0,C 180,E1 -17350.303,E2 -17350.303} C_VEL
LIN {X 0,Y 278.877,Z 602.868,A -85,B 0,C 180,E1 -17353.264,E2 -17353.264} C_VEL
LIN {X 0,Y 277.23,Z 609.054,A -85,B 0,C 180,E1 -17356.065,E2 -17356.065} C_VEL
LIN {X 0,Y 276.012,Z 613.938,A -85,B 0,C 180,E1 -17358.991,E2 -17358.991} C_VEL
LIN {X 0,Y 275.59,Z 616.673,A -85,B 0,C 180,E1 -17361.199,E2 -17361.199} C_VEL
LIN {X 0,Y 275.343,Z 619.145,A -85,B 0,C 180,E1 -17364.14,E2 -17364.14} C_VEL
LIN {X 0,Y 275.43,Z 620.252,A -85,B 0,C 180,E1 -17367.075,E2 -17367.075} C_VEL
LIN {X 0,Y 275.715,Z 619.982,A -85,B 0,C 180,E1 -17370,E2 -17370} C_VEL
LIN {X 0,Y 275.482,Z 618.232,A -85,B 0,C 180,E1 -17372.925,E2 -17372.925} C_VEL
LIN {X 0,Y 275.549,Z 616.804,A -85,B 0,C 180,E1 -17374.388,E2 -17374.388} C_VEL
LIN {X 0,Y 275.558,Z 614.026,A -85,B 0,C 180,E1 -17376.517,E2 -17376.517} C_VEL
LIN {X 0,Y 275.697,Z 610.117,A -85,B 0,C 180,E1 -17378.798,E2 -17378.798} C_VEL
LIN {X 0,Y 276.042,Z 605.359,A -85,B 0,C 180,E1 -17381.008,E2 -17381.008} C_VEL
LIN {X 0,Y 276.845,Z 598.423,A -85,B 0,C 180,E1 -17383.581,E2 -17383.581} C_VEL
LIN {X 0,Y 277.99,Z 589.789,A -85,B 0,C 180,E1 -17386.146,E2 -17386.146} C_VEL
LIN {X 0,Y 279.427,Z 580.808,A -85,B 0,C 180,E1 -17388.324,E2 -17388.324} C_VEL
LIN {X 0,Y 281.133,Z 569.984,A -85,B 0,C 180,E1 -17390.486,E2 -17390.486} C_VEL
LIN {X 0,Y 282.989,Z 559.162,A -85,B 0,C 180,E1 -17392.255,E2 -17392.255} C_VEL
LIN {X 0,Y 284.72,Z 548.087,A -85,B 0,C 180,E1 -17393.753,E2 -17393.753} C_VEL
LIN {X 0,Y 285.03,Z 544.596,A -85,B 0,C 180,E1 -17394.174,E2 -17394.174} C_VEL
LIN {X 0,Y 283.735,Z 531.498,A -85,B 0,C 180,E1 -17395.702,E2 -17395.702} C_VEL
LIN {X 0,Y 282.004,Z 518.237,A -85,B 0,C 180,E1 -17397.004,E2 -17397.004} C_VEL
LIN {X 0,Y 279.676,Z 502.981,A -85,B 0,C 180,E1 -17398.226,E2 -17398.226} C_VEL
LIN {X 0,Y 277.426,Z 490.104,A -85,B 0,C 180,E1 -17399.082,E2 -17399.082} C_VEL
LIN {X 0,Y 278.259,Z 484.778,A -85,B 0,C 180,E1 -17402.826,E2 -17402.826} C_VEL
LIN {X 0,Y 279.137,Z 479.899,A -85,B 0,C 180,E1 -17406.324,E2 -17406.324} C_VEL
LIN {X 0,Y 279.679,Z 476.365,A -85,B 0,C 180,E1 -17408.918,E2 -17408.918} C_VEL
LIN {X 0,Y 279.698,Z 473.52,A -85,B 0,C 180,E1 -17411.078,E2 -17411.078} C_VEL
LIN {X 0,Y 278.968,Z 468.83,A -85,B 0,C 180,E1 -17414.861,E2 -17414.861} C_VEL
LIN {X 0,Y 277.988,Z 463.595,A -85,B 0,C 180,E1 -17419.327,E2 -17419.327} C_VEL
LIN {X 0,Y 277.36,Z 459.564,A -85,B 0,C 180,E1 -17422.994,E2 -17422.994} C_VEL
LIN {X 0,Y 277.242,Z 459.573,A -85,B 0,C 180,E1 -17427.836,E2 -17427.836} C_VEL
LIN {X 0,Y 277.286,Z 459.57,A -85,B 0,C 180,E1 -17431.212,E2 -17431.212} C_VEL
LIN {X 0,Y 277.31,Z 459.564,A -85,B 0,C 180,E1 -17434.479,E2 -17434.479} C_VEL
LIN {X 0,Y 277.281,Z 459.568,A -85,B 0,C 180,E1 -17437.655,E2 -17437.655} C_VEL
LIN {X 0,Y 277.341,Z 459.565,A -85,B 0,C 180,E1 -17440.766,E2 -17440.766} C_VEL
LIN {X 0,Y 277.43,Z 459.55,A -85,B 0,C 180,E1 -17445.326,E2 -17445.326} C_VEL
LIN {X 0,Y 277.502,Z 459.54,A -85,B 0,C 180,E1 -17449.789,E2 -17449.789} C_VEL
LIN {X 0,Y 277.648,Z 459.525,A -85,B 0,C 180,E1 -17452.729,E2 -17452.729} C_VEL
LIN {X 0,Y 277.818,Z 459.506,A -85,B 0,C 180,E1 -17458.551,E2 -17458.551} C_VEL
LIN {X 0,Y 277.82,Z 459.499,A -85,B 0,C 180,E1 -17461.45,E2 -17461.45} C_VEL
LIN {X 0,Y 277.65,Z 459.522,A -85,B 0,C 180,E1 -17467.271,E2 -17467.271} C_VEL
LIN {X 0,Y 277.503,Z 459.542,A -85,B 0,C 180,E1 -17470.212,E2 -17470.212} C_VEL
LIN {X 0,Y 277.424,Z 459.553,A -85,B 0,C 180,E1 -17474.675,E2 -17474.675} C_VEL
LIN {X 0,Y 277.342,Z 459.559,A -85,B 0,C 180,E1 -17479.234,E2 -17479.234} C_VEL
LIN {X 0,Y 277.316,Z 459.568,A -85,B 0,C 180,E1 -17484.171,E2 -17484.171} C_VEL
LIN {X 0,Y 277.323,Z 459.562,A -85,B 0,C 180,E1 -17487.506,E2 -17487.506} C_VEL
LIN {X 0,Y 277.27,Z 459.572,A -85,B 0,C 180,E1 -17490.482,E2 -17490.482} C_VEL
LIN {X 0,Y 277.245,Z 459.575,A -85,B 0,C 180,E1 -17493.896,E2 -17493.896} C_VEL
LIN {X 0,Y 277.27,Z 459.568,A -85,B 0,C 180,E1 -17497.469,E2 -17497.469} C_VEL
LIN {X 0,Y 277.208,Z 459.577,A -85,B 0,C 180,E1 -17501.237,E2 -17501.237} C_VEL
LIN {X 0,Y 277.206,Z 459.576,A -85,B 0,C 180,E1 -17505.226,E2 -17505.226} C_VEL
LIN {X 0,Y 277.262,Z 459.572,A -85,B 0,C 180,E1 -17509.503,E2 -17509.503} C_VEL
LIN {X 0,Y 277.288,Z 459.567,A -85,B 0,C 180,E1 -17512.535,E2 -17512.535} C_VEL
LIN {X 0,Y 277.255,Z 459.574,A -85,B 0,C 180,E1 -17516.106,E2 -17516.106} C_VEL
LIN {X 0,Y 277.263,Z 459.573,A -85,B 0,C 180,E1 -17519.539,E2 -17519.539} C_VEL
LIN {X 0,Y 277.364,Z 459.556,A -85,B 0,C 180,E1 -17522.865,E2 -17522.865} C_VEL
LIN {X 0,Y 277.331,Z 459.564,A -85,B 0,C 180,E1 -17526.08,E2 -17526.08} C_VEL
LIN {X 0,Y 277.348,Z 459.559,A -85,B 0,C 180,E1 -17530.767,E2 -17530.767} C_VEL
LIN {X 0,Y 277.438,Z 459.551,A -85,B 0,C 180,E1 -17535.326,E2 -17535.326} C_VEL
LIN {X 0,Y 277.463,Z 459.547,A -85,B 0,C 180,E1 -17539.787,E2 -17539.787} C_VEL
LIN {X 0,Y 277.609,Z 459.527,A -85,B 0,C 180,E1 -17542.728,E2 -17542.728} C_VEL
LIN {X 0,Y 277.824,Z 459.5,A -85,B 0,C 180,E1 -17548.55,E2 -17548.55} C_VEL
LIN {X 0,Y 277.824,Z 459.504,A -85,B 0,C 180,E1 -17551.45,E2 -17551.45} C_VEL
LIN {X 0,Y 277.644,Z 459.527,A -85,B 0,C 180,E1 -17557.271,E2 -17557.271} C_VEL
LIN {X 0,Y 277.464,Z 459.543,A -85,B 0,C 180,E1 -17560.213,E2 -17560.213} C_VEL
LIN {X 0,Y 277.438,Z 459.55,A -85,B 0,C 180,E1 -17564.674,E2 -17564.674} C_VEL
LIN {X 0,Y 277.348,Z 459.564,A -85,B 0,C 180,E1 -17569.233,E2 -17569.233} C_VEL
LIN {X 0,Y 277.321,Z 459.563,A -85,B 0,C 180,E1 -17574.17,E2 -17574.17} C_VEL
LIN {X 0,Y 277.327,Z 459.564,A -85,B 0,C 180,E1 -17577.505,E2 -17577.505} C_VEL
LIN {X 0,Y 277.273,Z 459.571,A -85,B 0,C 180,E1 -17580.481,E2 -17580.481} C_VEL
LIN {X 0,Y 277.126,Z 459.588,A -85,B 0,C 180,E1 -17583.912,E2 -17583.912} C_VEL
LIN {X 0,Y 276.838,Z 459.624,A -85,B 0,C 180,E1 -17587.537,E2 -17587.537} C_VEL
LIN {X 0,Y 276.369,Z 459.686,A -85,B 0,C 180,E1 -17591.389,E2 -17591.389} C_VEL
LIN {X 0,Y 276.18,Z 459.71,A -85,B 0,C 180,E1 -17593.069,E2 -17593.069} C_VEL
LIN {X 0,Y 280.781,Z 475.66,A -85,B 0,C 180,E1 -17594.334,E2 -17594.334} C_VEL
LIN {X 0,Y 284.205,Z 488.871,A -85,B 0,C 180,E1 -17595.593,E2 -17595.593} C_VEL
LIN {X 0,Y 287.053,Z 501.363,A -85,B 0,C 180,E1 -17596.981,E2 -17596.981} C_VEL
LIN {X 0,Y 287.318,Z 503.284,A -85,B 0,C 180,E1 -17597.207,E2 -17597.207} C_VEL
LIN {X 0,Y 285.43,Z 517.282,A -85,B 0,C 180,E1 -17598.802,E2 -17598.802} C_VEL
LIN {X 0,Y 283.577,Z 529.958,A -85,B 0,C 180,E1 -17600.603,E2 -17600.603} C_VEL
LIN {X 0,Y 281.882,Z 540.569,A -85,B 0,C 180,E1 -17602.439,E2 -17602.439} C_VEL
LIN {X 0,Y 280.397,Z 549.806,A -85,B 0,C 180,E1 -17604.355,E2 -17604.355} C_VEL
LIN {X 0,Y 278.776,Z 559.367,A -85,B 0,C 180,E1 -17606.748,E2 -17606.748} C_VEL
LIN {X 0,Y 277.77,Z 566.033,A -85,B 0,C 180,E1 -17608.756,E2 -17608.756} C_VEL
LIN {X 0,Y 276.897,Z 572.655,A -85,B 0,C 180,E1 -17611.168,E2 -17611.168} C_VEL
LIN {X 0,Y 276.189,Z 578.08,A -85,B 0,C 180,E1 -17613.622,E2 -17613.622} C_VEL
LIN {X 0,Y 275.733,Z 582.081,A -85,B 0,C 180,E1 -17615.932,E2 -17615.932} C_VEL
LIN {X 0,Y 275.474,Z 584.273,A -85,B 0,C 180,E1 -17617.499,E2 -17617.499} C_VEL
LIN {X 0,Y 275.315,Z 586.046,A -85,B 0,C 180,E1 -17619.06,E2 -17619.06} C_VEL
LIN {X 0,Y 275.292,Z 587.54,A -85,B 0,C 180,E1 -17620.833,E2 -17620.833} C_VEL
LIN {X 0,Y 275.377,Z 588.922,A -85,B 0,C 180,E1 -17623.696,E2 -17623.696} C_VEL
LIN {X 0,Y 275.82,Z 588.983,A -85,B 0,C 180,E1 -17626.742,E2 -17626.742} C_VEL
LIN {X 0,Y 276.584,Z 587.646,A -85,B 0,C 180,E1 -17629.754,E2 -17629.754} C_VEL
LIN {X 0,Y 277.84,Z 584.925,A -85,B 0,C 180,E1 -17632.734,E2 -17632.734} C_VEL
LIN {X 0,Y 279.511,Z 580.791,A -85,B 0,C 180,E1 -17635.674,E2 -17635.674} C_VEL
LIN {X 0,Y 281.816,Z 575.08,A -85,B 0,C 180,E1 -17638.571,E2 -17638.571} C_VEL
LIN {X 0,Y 284.629,Z 567.717,A -85,B 0,C 180,E1 -17641.415,E2 -17641.415} C_VEL
LIN {X 0,Y 287.64,Z 559.654,A -85,B 0,C 180,E1 -17643.852,E2 -17643.852} C_VEL
LIN {X 0,Y 290.668,Z 551.364,A -85,B 0,C 180,E1 -17645.898,E2 -17645.898} C_VEL
LIN {X 0,Y 293.985,Z 541.525,A -85,B 0,C 180,E1 -17647.901,E2 -17647.901} C_VEL
LIN {X 0,Y 295.833,Z 535.677,A -85,B 0,C 180,E1 -17648.919,E2 -17648.919} C_VEL
LIN {X 0,Y 296.673,Z 531.352,A -85,B 0,C 180,E1 -17649.69,E2 -17649.69} C_VEL
LIN {X 0,Y 296.748,Z 527.215,A -85,B 0,C 180,E1 -17650.527,E2 -17650.527} C_VEL
LIN {X 0,Y 296.479,Z 524.565,A -85,B 0,C 180,E1 -17651.106,E2 -17651.106} C_VEL
LIN {X 0,Y 294.199,Z 514.31,A -85,B 0,C 180,E1 -17653.504,E2 -17653.504} C_VEL
LIN {X 0,Y 291.81,Z 505.741,A -85,B 0,C 180,E1 -17655.561,E2 -17655.561} C_VEL
LIN {X 0,Y 289.039,Z 498.4,A -85,B 0,C 180,E1 -17657.541,E2 -17657.541} C_VEL
LIN {X 0,Y 285.531,Z 491.198,A -85,B 0,C 180,E1 -17659.835,E2 -17659.835} C_VEL
LIN {X 0,Y 283.224,Z 487.04,A -85,B 0,C 180,E1 -17661.4,E2 -17661.4} C_VEL
LIN {X 0,Y 281.451,Z 484.933,A -85,B 0,C 180,E1 -17662.498,E2 -17662.498} C_VEL
LIN {X 0,Y 279.674,Z 482.015,A -85,B 0,C 180,E1 -17663.849,E2 -17663.849} C_VEL
LIN {X 0,Y 277.507,Z 479.59,A -85,B 0,C 180,E1 -17665.501,E2 -17665.501} C_VEL
LIN {X 0,Y 276.683,Z 477.675,A -85,B 0,C 180,E1 -17666.393,E2 -17666.393} C_VEL
LIN {X 0,Y 273.736,Z 475.831,A -85,B 0,C 180,E1 -17669.201,E2 -17669.201} C_VEL
LIN {X 0,Y 272.474,Z 473.475,A -85,B 0,C 180,E1 -17671.662,E2 -17671.662} C_VEL
LIN {X 0,Y 272.622,Z 474.329,A -85,B 0,C 180,E1 -17674.551,E2 -17674.551} C_VEL
LIN {X 0,Y 272.905,Z 475.806,A -85,B 0,C 180,E1 -17678.174,E2 -17678.174} C_VEL
LIN {X 0,Y 273.274,Z 477.667,A -85,B 0,C 180,E1 -17681.347,E2 -17681.347} C_VEL
LIN {X 0,Y 275.637,Z 483.19,A -85,B 0,C 180,E1 -17684.446,E2 -17684.446} C_VEL
LIN {X 0,Y 278.011,Z 486.319,A -85,B 0,C 180,E1 -17686.322,E2 -17686.322} C_VEL
LIN {X 0,Y 279.372,Z 490.169,A -85,B 0,C 180,E1 -17687.591,E2 -17687.591} C_VEL
LIN {X 0,Y 281.083,Z 493.122,A -85,B 0,C 180,E1 -17688.773,E2 -17688.773} C_VEL
LIN {X 0,Y 282.084,Z 496.348,A -85,B 0,C 180,E1 -17689.626,E2 -17689.626} C_VEL
LIN {X 0,Y 283.147,Z 498.383,A -85,B 0,C 180,E1 -17690.305,E2 -17690.305} C_VEL
LIN {X 0,Y 285.959,Z 508.186,A -85,B 0,C 180,E1 -17692.597,E2 -17692.597} C_VEL
LIN {X 0,Y 287.949,Z 517.182,A -85,B 0,C 180,E1 -17694.45,E2 -17694.45} C_VEL
LIN {X 0,Y 289.475,Z 528.352,A -85,B 0,C 180,E1 -17696.518,E2 -17696.518} C_VEL
LIN {X 0,Y 289.941,Z 539.736,A -85,B 0,C 180,E1 -17698.501,E2 -17698.501} C_VEL
LIN {X 0,Y 289.299,Z 549.476,A -85,B 0,C 180,E1 -17700.132,E2 -17700.132} C_VEL
LIN {X 0,Y 288.228,Z 556.132,A -85,B 0,C 180,E1 -17701.252,E2 -17701.252} C_VEL
LIN {X 0,Y 284.248,Z 567.805,A -85,B 0,C 180,E1 -17703.175,E2 -17703.175} C_VEL
LIN {X 0,Y 280.785,Z 577.898,A -85,B 0,C 180,E1 -17705.213,E2 -17705.213} C_VEL
LIN {X 0,Y 277.31,Z 587.774,A -85,B 0,C 180,E1 -17707.657,E2 -17707.657} C_VEL
LIN {X 0,Y 274.072,Z 597.03,A -85,B 0,C 180,E1 -17710.528,E2 -17710.528} C_VEL
LIN {X 0,Y 271.644,Z 604.498,A -85,B 0,C 180,E1 -17713.466,E2 -17713.466} C_VEL
LIN {X 0,Y 269.918,Z 610.377,A -85,B 0,C 180,E1 -17716.448,E2 -17716.448} C_VEL
LIN {X 0,Y 268.811,Z 614.797,A -85,B 0,C 180,E1 -17719.455,E2 -17719.455} C_VEL
LIN {X 0,Y 268.316,Z 617.821,A -85,B 0,C 180,E1 -17722.475,E2 -17722.475} C_VEL
LIN {X 0,Y 268.274,Z 619.498,A -85,B 0,C 180,E1 -17725.492,E2 -17725.492} C_VEL
LIN {X 0,Y 268.354,Z 619.824,A -85,B 0,C 180,E1 -17726.998,E2 -17726.998} C_VEL
LIN {X 0,Y 268.631,Z 619.429,A -85,B 0,C 180,E1 -17730,E2 -17730} C_VEL
LIN {X 0,Y 268.412,Z 617.559,A -85,B 0,C 180,E1 -17733.002,E2 -17733.002} C_VEL
LIN {X 0,Y 268.491,Z 616.085,A -85,B 0,C 180,E1 -17734.504,E2 -17734.504} C_VEL
LIN {X 0,Y 268.497,Z 613.157,A -85,B 0,C 180,E1 -17736.764,E2 -17736.764} C_VEL
LIN {X 0,Y 268.642,Z 609.253,A -85,B 0,C 180,E1 -17739.031,E2 -17739.031} C_VEL
LIN {X 0,Y 269.041,Z 604.377,A -85,B 0,C 180,E1 -17741.298,E2 -17741.298} C_VEL
LIN {X 0,Y 269.876,Z 597.307,A -85,B 0,C 180,E1 -17743.938,E2 -17743.938} C_VEL
LIN {X 0,Y 270.959,Z 589.415,A -85,B 0,C 180,E1 -17746.324,E2 -17746.324} C_VEL
LIN {X 0,Y 272.602,Z 579.383,A -85,B 0,C 180,E1 -17748.8,E2 -17748.8} C_VEL
LIN {X 0,Y 274.416,Z 568.324,A -85,B 0,C 180,E1 -17751.011,E2 -17751.011} C_VEL
LIN {X 0,Y 276.276,Z 557.211,A -85,B 0,C 180,E1 -17752.826,E2 -17752.826} C_VEL
LIN {X 0,Y 278.005,Z 546.807,A -85,B 0,C 180,E1 -17754.239,E2 -17754.239} C_VEL
LIN {X 0,Y 277.13,Z 535.281,A -85,B 0,C 180,E1 -17755.679,E2 -17755.679} C_VEL
LIN {X 0,Y 275.37,Z 520.701,A -85,B 0,C 180,E1 -17757.218,E2 -17757.218} C_VEL
LIN {X 0,Y 273.092,Z 505.08,A -85,B 0,C 180,E1 -17758.562,E2 -17758.562} C_VEL
LIN {X 0,Y 270.441,Z 489.805,A -85,B 0,C 180,E1 -17759.587,E2 -17759.587} C_VEL
LIN {X 0,Y 271.198,Z 485.141,A -85,B 0,C 180,E1 -17762.97,E2 -17762.97} C_VEL
LIN {X 0,Y 272.183,Z 479.893,A -85,B 0,C 180,E1 -17766.828,E2 -17766.828} C_VEL
LIN {X 0,Y 272.659,Z 476.565,A -85,B 0,C 180,E1 -17769.352,E2 -17769.352} C_VEL
LIN {X 0,Y 272.5,Z 473.102,A -85,B 0,C 180,E1 -17772.11,E2 -17772.11} C_VEL
LIN {X 0,Y 271.588,Z 467.952,A -85,B 0,C 180,E1 -17776.432,E2 -17776.432} C_VEL
LIN {X 0,Y 270.655,Z 462.657,A -85,B 0,C 180,E1 -17781.168,E2 -17781.168} C_VEL
LIN {X 0,Y 270.291,Z 460.445,A -85,B 0,C 180,E1 -17783.271,E2 -17783.271} C_VEL
LIN {X 0,Y 270.202,Z 460.452,A -85,B 0,C 180,E1 -17786.893,E2 -17786.893} C_VEL
LIN {X 0,Y 270.225,Z 460.448,A -85,B 0,C 180,E1 -17790.386,E2 -17790.386} C_VEL
LIN {X 0,Y 270.26,Z 460.441,A -85,B 0,C 180,E1 -17793.764,E2 -17793.764} C_VEL
LIN {X 0,Y 270.229,Z 460.45,A -85,B 0,C 180,E1 -17797.039,E2 -17797.039} C_VEL
LIN {X 0,Y 270.297,Z 460.439,A -85,B 0,C 180,E1 -17800.244,E2 -17800.244} C_VEL
LIN {X 0,Y 270.399,Z 460.428,A -85,B 0,C 180,E1 -17804.935,E2 -17804.935} C_VEL
LIN {X 0,Y 270.437,Z 460.421,A -85,B 0,C 180,E1 -17809.519,E2 -17809.519} C_VEL
LIN {X 0,Y 270.606,Z 460.402,A -85,B 0,C 180,E1 -17812.539,E2 -17812.539} C_VEL
LIN {X 0,Y 270.784,Z 460.381,A -85,B 0,C 180,E1 -17818.513,E2 -17818.513} C_VEL
LIN {X 0,Y 270.786,Z 460.375,A -85,B 0,C 180,E1 -17821.488,E2 -17821.488} C_VEL
LIN {X 0,Y 270.608,Z 460.399,A -85,B 0,C 180,E1 -17827.462,E2 -17827.462} C_VEL
LIN {X 0,Y 270.438,Z 460.423,A -85,B 0,C 180,E1 -17830.482,E2 -17830.482} C_VEL
LIN {X 0,Y 270.393,Z 460.427,A -85,B 0,C 180,E1 -17835.066,E2 -17835.066} C_VEL
LIN {X 0,Y 270.298,Z 460.437,A -85,B 0,C 180,E1 -17839.756,E2 -17839.756} C_VEL
LIN {X 0,Y 270.271,Z 460.443,A -85,B 0,C 180,E1 -17844.586,E2 -17844.586} C_VEL
LIN {X 0,Y 270.27,Z 460.443,A -85,B 0,C 180,E1 -17847.909,E2 -17847.909} C_VEL
LIN {X 0,Y 270.182,Z 460.452,A -85,B 0,C 180,E1 -17851.349,E2 -17851.349} C_VEL
LIN {X 0,Y 270.2,Z 460.45,A -85,B 0,C 180,E1 -17854.906,E2 -17854.906} C_VEL
LIN {X 0,Y 270.196,Z 460.451,A -85,B 0,C 180,E1 -17858.711,E2 -17858.711} C_VEL
LIN {X 0,Y 270.171,Z 460.455,A -85,B 0,C 180,E1 -17862.559,E2 -17862.559} C_VEL
LIN {X 0,Y 270.18,Z 460.452,A -85,B 0,C 180,E1 -17866.748,E2 -17866.748} C_VEL
LIN {X 0,Y 270.213,Z 460.45,A -85,B 0,C 180,E1 -17869.442,E2 -17869.442} C_VEL
LIN {X 0,Y 270.257,Z 460.446,A -85,B 0,C 180,E1 -17873.722,E2 -17873.722} C_VEL
LIN {X 0,Y 270.205,Z 460.449,A -85,B 0,C 180,E1 -17876.894,E2 -17876.894} C_VEL
LIN {X 0,Y 270.238,Z 460.446,A -85,B 0,C 180,E1 -17880.388,E2 -17880.388} C_VEL
LIN {X 0,Y 270.268,Z 460.444,A -85,B 0,C 180,E1 -17883.765,E2 -17883.765} C_VEL
LIN {X 0,Y 270.235,Z 460.446,A -85,B 0,C 180,E1 -17887.039,E2 -17887.039} C_VEL
LIN {X 0,Y 270.304,Z 460.437,A -85,B 0,C 180,E1 -17890.245,E2 -17890.245} C_VEL
LIN {X 0,Y 270.406,Z 460.425,A -85,B 0,C 180,E1 -17894.936,E2 -17894.936} C_VEL
LIN {X 0,Y 270.415,Z 460.427,A -85,B 0,C 180,E1 -17899.518,E2 -17899.518} C_VEL
LIN {X 0,Y 270.57,Z 460.403,A -85,B 0,C 180,E1 -17902.538,E2 -17902.538} C_VEL
LIN {X 0,Y 270.79,Z 460.376,A -85,B 0,C 180,E1 -17908.513,E2 -17908.513} C_VEL
LIN {X 0,Y 270.79,Z 460.38,A -85,B 0,C 180,E1 -17911.487,E2 -17911.487} C_VEL
LIN {X 0,Y 270.602,Z 460.402,A -85,B 0,C 180,E1 -17917.461,E2 -17917.461} C_VEL
LIN {X 0,Y 270.416,Z 460.422,A -85,B 0,C 180,E1 -17920.482,E2 -17920.482} C_VEL
LIN {X 0,Y 270.406,Z 460.429,A -85,B 0,C 180,E1 -17925.064,E2 -17925.064} C_VEL
LIN {X 0,Y 270.304,Z 460.438,A -85,B 0,C 180,E1 -17929.755,E2 -17929.755} C_VEL
LIN {X 0,Y 270.276,Z 460.442,A -85,B 0,C 180,E1 -17934.585,E2 -17934.585} C_VEL
LIN {X 0,Y 270.274,Z 460.442,A -85,B 0,C 180,E1 -17937.908,E2 -17937.908} C_VEL
LIN {X 0,Y 270.17,Z 460.456,A -85,B 0,C 180,E1 -17941.349,E2 -17941.349} C_VEL
LIN {X 0,Y 270.021,Z 460.477,A -85,B 0,C 180,E1 -17944.931,E2 -17944.931} C_VEL
LIN {X 0,Y 269.633,Z 460.525,A -85,B 0,C 180,E1 -17948.723,E2 -17948.723} C_VEL
LIN {X 0,Y 269.2,Z 460.579,A -85,B 0,C 180,E1 -17952.557,E2 -17952.557} C_VEL
LIN {X 0,Y 273.839,Z 476.395,A -85,B 0,C 180,E1 -17953.863,E2 -17953.863} C_VEL
LIN {X 0,Y 277.337,Z 490.028,A -85,B 0,C 180,E1 -17955.197,E2 -17955.197} C_VEL
LIN {X 0,Y 280.202,Z 502.687,A -85,B 0,C 180,E1 -17956.666,E2 -17956.666} C_VEL
LIN {X 0,Y 280.283,Z 505.449,A -85,B 0,C 180,E1 -17956.989,E2 -17956.989} C_VEL
LIN {X 0,Y 278.491,Z 518.277,A -85,B 0,C 180,E1 -17958.513,E2 -17958.513} C_VEL
LIN {X 0,Y 276.595,Z 530.859,A -85,B 0,C 180,E1 -17960.359,E2 -17960.359} C_VEL
LIN {X 0,Y 274.66,Z 542.594,A -85,B 0,C 180,E1 -17962.487,E2 -17962.487} C_VEL
LIN {X 0,Y 273.068,Z 552.242,A -85,B 0,C 180,E1 -17964.613,E2 -17964.613} C_VEL
LIN {X 0,Y 271.462,Z 561.417,A -85,B 0,C 180,E1 -17967.065,E2 -17967.065} C_VEL
LIN {X 0,Y 270.299,Z 569.357,A -85,B 0,C 180,E1 -17969.681,E2 -17969.681} C_VEL
LIN {X 0,Y 269.364,Z 576.213,A -85,B 0,C 180,E1 -17972.509,E2 -17972.509} C_VEL
LIN {X 0,Y 268.751,Z 581.369,A -85,B 0,C 180,E1 -17975.265,E2 -17975.265} C_VEL
LIN {X 0,Y 268.478,Z 583.747,A -85,B 0,C 180,E1 -17976.88,E2 -17976.88} C_VEL
LIN {X 0,Y 268.181,Z 587.237,A -85,B 0,C 180,E1 -17980.081,E2 -17980.081} C_VEL
LIN {X 0,Y 268.275,Z 589.159,A -85,B 0,C 180,E1 -17983.251,E2 -17983.251} C_VEL
LIN {X 0,Y 268.682,Z 589.6,A -85,B 0,C 180,E1 -17986.384,E2 -17986.384} C_VEL
LIN {X 0,Y 269.413,Z 588.617,A -85,B 0,C 180,E1 -17989.478,E2 -17989.478} C_VEL
LIN {X 0,Y 270.669,Z 586.218,A -85,B 0,C 180,E1 -17992.54,E2 -17992.54} C_VEL
LIN {X 0,Y 272.34,Z 582.448,A -85,B 0,C 180,E1 -17995.56,E2 -17995.56} C_VEL
LIN {X 0,Y 274.716,Z 577.173,A -85,B 0,C 180,E1 -17998.534,E2 -17998.534} C_VEL
LIN {X 0,Y 277.583,Z 570.298,A -85,B 0,C 180,E1 -18001.451,E2 -18001.451} C_VEL
LIN {X 0,Y 280.652,Z 562.791,A -85,B 0,C 180,E1 -18003.949,E2 -18003.949} C_VEL
LIN {X 0,Y 284.284,Z 553.519,A -85,B 0,C 180,E1 -18006.387,E2 -18006.387} C_VEL
LIN {X 0,Y 288.354,Z 542.281,A -85,B 0,C 180,E1 -18008.762,E2 -18008.762} C_VEL
LIN {X 0,Y 291.928,Z 531.63,A -85,B 0,C 180,E1 -18010.577,E2 -18010.577} C_VEL
LIN {X 0,Y 295.009,Z 521.298,A -85,B 0,C 180,E1 -18012.032,E2 -18012.032} C_VEL
LIN {X 0,Y 295.029,Z 519.262,A -85,B 0,C 180,E1 -18012.404,E2 -18012.404} C_VEL
LIN {X 0,Y 294.199,Z 514.31,A -85,B 0,C 180,E1 -18013.504,E2 -18013.504} C_VEL
LIN {X 0,Y 292.827,Z 511.015,A -85,B 0,C 180,E1 -18014.42,E2 -18014.42} C_VEL
LIN {X 0,Y 290.771,Z 508.503,A -85,B 0,C 180,E1 -18015.397,E2 -18015.397} C_VEL
LIN {X 0,Y 284.723,Z 502.818,A -85,B 0,C 180,E1 -18018.136,E2 -18018.136} C_VEL
LIN {X 0,Y 283.633,Z 500.977,A -85,B 0,C 180,E1 -18018.821,E2 -18018.821} C_VEL
LIN {X 0,Y 280.38,Z 494.34,A -85,B 0,C 180,E1 -18021.271,E2 -18021.271} C_VEL
LIN {X 0,Y 279.146,Z 492.232,A -85,B 0,C 180,E1 -18022.188,E2 -18022.188} C_VEL
LIN {X 0,Y 276.931,Z 488.525,A -85,B 0,C 180,E1 -18023.993,E2 -18023.993} C_VEL
LIN {X 0,Y 274.832,Z 486.027,A -85,B 0,C 180,E1 -18025.768,E2 -18025.768} C_VEL
LIN {X 0,Y 274.382,Z 484.972,A -85,B 0,C 180,E1 -18026.302,E2 -18026.302} C_VEL
LIN {X 0,Y 271.475,Z 482.461,A -85,B 0,C 180,E1 -18029.464,E2 -18029.464} C_VEL
LIN {X 0,Y 270.613,Z 480.709,A -85,B 0,C 180,E1 -18031.293,E2 -18031.293} C_VEL
LIN {X 0,Y 269.672,Z 480.502,A -85,B 0,C 180,E1 -18033.494,E2 -18033.494} C_VEL
LIN {X 0,Y 269.428,Z 481.564,A -85,B 0,C 180,E1 -18037.1,E2 -18037.1} C_VEL
LIN {X 0,Y 271.052,Z 484.11,A -85,B 0,C 180,E1 -18040.929,E2 -18040.929} C_VEL
LIN {X 0,Y 273.054,Z 489.49,A -85,B 0,C 180,E1 -18044.022,E2 -18044.022} C_VEL
LIN {X 0,Y 274.96,Z 492.06,A -85,B 0,C 180,E1 -18045.699,E2 -18045.699} C_VEL
LIN {X 0,Y 275.966,Z 495.589,A -85,B 0,C 180,E1 -18046.917,E2 -18046.917} C_VEL
LIN {X 0,Y 277.301,Z 497.974,A -85,B 0,C 180,E1 -18047.936,E2 -18047.936} C_VEL
LIN {X 0,Y 279.428,Z 504.229,A -85,B 0,C 180,E1 -18049.854,E2 -18049.854} C_VEL
LIN {X 0,Y 281.515,Z 512.695,A -85,B 0,C 180,E1 -18051.953,E2 -18051.953} C_VEL
LIN {X 0,Y 283.053,Z 520.979,A -85,B 0,C 180,E1 -18053.764,E2 -18053.764} C_VEL
LIN {X 0,Y 284.122,Z 531.343,A -85,B 0,C 180,E1 -18055.801,E2 -18055.801} C_VEL
LIN {X 0,Y 284.23,Z 543.001,A -85,B 0,C 180,E1 -18057.949,E2 -18057.949} C_VEL
LIN {X 0,Y 283.238,Z 552.456,A -85,B 0,C 180,E1 -18059.632,E2 -18059.632} C_VEL
LIN {X 0,Y 282.155,Z 557.844,A -85,B 0,C 180,E1 -18060.573,E2 -18060.573} C_VEL
LIN {X 0,Y 278.139,Z 568.867,A -85,B 0,C 180,E1 -18062.477,E2 -18062.477} C_VEL
LIN {X 0,Y 274.415,Z 578.813,A -85,B 0,C 180,E1 -18064.598,E2 -18064.598} C_VEL
LIN {X 0,Y 271.29,Z 587.166,A -85,B 0,C 180,E1 -18066.73,E2 -18066.73} C_VEL
LIN {X 0,Y 268.182,Z 595.363,A -85,B 0,C 180,E1 -18069.282,E2 -18069.282} C_VEL
LIN {X 0,Y 265.341,Z 603.013,A -85,B 0,C 180,E1 -18072.267,E2 -18072.267} C_VEL
LIN {X 0,Y 263.384,Z 609.086,A -85,B 0,C 180,E1 -18075.316,E2 -18075.316} C_VEL
LIN {X 0,Y 262.24,Z 612.696,A -85,B 0,C 180,E1 -18077.62,E2 -18077.62} C_VEL
LIN {X 0,Y 261.466,Z 616.259,A -85,B 0,C 180,E1 -18080.719,E2 -18080.719} C_VEL
LIN {X 0,Y 261.155,Z 618.476,A -85,B 0,C 180,E1 -18083.821,E2 -18083.821} C_VEL
LIN {X 0,Y 261.278,Z 619.355,A -85,B 0,C 180,E1 -18086.916,E2 -18086.916} C_VEL
LIN {X 0,Y 261.548,Z 618.853,A -85,B 0,C 180,E1 -18090,E2 -18090} C_VEL
LIN {X 0,Y 261.345,Z 616.875,A -85,B 0,C 180,E1 -18093.083,E2 -18093.083} C_VEL
LIN {X 0,Y 261.433,Z 615.342,A -85,B 0,C 180,E1 -18094.626,E2 -18094.626} C_VEL
LIN {X 0,Y 261.44,Z 612.311,A -85,B 0,C 180,E1 -18096.948,E2 -18096.948} C_VEL
LIN {X 0,Y 261.601,Z 608.322,A -85,B 0,C 180,E1 -18099.276,E2 -18099.276} C_VEL
LIN {X 0,Y 262.023,Z 603.324,A -85,B 0,C 180,E1 -18101.605,E2 -18101.605} C_VEL
LIN {X 0,Y 262.899,Z 596.126,A -85,B 0,C 180,E1 -18104.316,E2 -18104.316} C_VEL
LIN {X 0,Y 263.952,Z 588.826,A -85,B 0,C 180,E1 -18106.557,E2 -18106.557} C_VEL
LIN {X 0,Y 265.532,Z 579.544,A -85,B 0,C 180,E1 -18108.918,E2 -18108.918} C_VEL
LIN {X 0,Y 267.359,Z 568.668,A -85,B 0,C 180,E1 -18111.188,E2 -18111.188} C_VEL
LIN {X 0,Y 269.258,Z 557.747,A -85,B 0,C 180,E1 -18113.049,E2 -18113.049} C_VEL
LIN {X 0,Y 271.019,Z 547.372,A -85,B 0,C 180,E1 -18114.513,E2 -18114.513} C_VEL
LIN {X 0,Y 270.173,Z 535.559,A -85,B 0,C 180,E1 -18116.044,E2 -18116.044} C_VEL
LIN {X 0,Y 268.627,Z 522.476,A -85,B 0,C 180,E1 -18117.492,E2 -18117.492} C_VEL
LIN {X 0,Y 266.424,Z 506.949,A -85,B 0,C 180,E1 -18118.894,E2 -18118.894} C_VEL
LIN {X 0,Y 263.706,Z 491.362,A -85,B 0,C 180,E1 -18120.018,E2 -18120.018} C_VEL
LIN {X 0,Y 263.472,Z 489.436,A -85,B 0,C 180,E1 -18120.147,E2 -18120.147} C_VEL
LIN {X 0,Y 264.533,Z 483.561,A -85,B 0,C 180,E1 -18124.554,E2 -18124.554} C_VEL
LIN {X 0,Y 265.479,Z 478.463,A -85,B 0,C 180,E1 -18128.47,E2 -18128.47} C_VEL
LIN {X 0,Y 265.639,Z 476.659,A -85,B 0,C 180,E1 -18129.893,E2 -18129.893} C_VEL
LIN {X 0,Y 265.439,Z 473.889,A -85,B 0,C 180,E1 -18132.153,E2 -18132.153} C_VEL
LIN {X 0,Y 264.575,Z 469.065,A -85,B 0,C 180,E1 -18136.319,E2 -18136.319} C_VEL
LIN {X 0,Y 263.741,Z 464.376,A -85,B 0,C 180,E1 -18140.602,E2 -18140.602} C_VEL
LIN {X 0,Y 263.233,Z 461.324,A -85,B 0,C 180,E1 -18143.61,E2 -18143.61} C_VEL
LIN {X 0,Y 263.131,Z 461.332,A -85,B 0,C 180,E1 -18147.712,E2 -18147.712} C_VEL
LIN {X 0,Y 263.198,Z 461.322,A -85,B 0,C 180,E1 -18151.783,E2 -18151.783} C_VEL
LIN {X 0,Y 263.222,Z 461.32,A -85,B 0,C 180,E1 -18155.2,E2 -18155.2} C_VEL
LIN {X 0,Y 263.26,Z 461.315,A -85,B 0,C 180,E1 -18159.693,E2 -18159.693} C_VEL
LIN {X 0,Y 263.347,Z 461.304,A -85,B 0,C 180,E1 -18164.522,E2 -18164.522} C_VEL
LIN {X 0,Y 263.37,Z 461.302,A -85,B 0,C 180,E1 -18169.235,E2 -18169.235} C_VEL
LIN {X 0,Y 263.568,Z 461.277,A -85,B 0,C 180,E1 -18172.339,E2 -18172.339} C_VEL
LIN {X 0,Y 263.748,Z 461.257,A -85,B 0,C 180,E1 -18178.473,E2 -18178.473} C_VEL
LIN {X 0,Y 263.75,Z 461.252,A -85,B 0,C 180,E1 -18181.527,E2 -18181.527} C_VEL
LIN {X 0,Y 263.57,Z 461.276,A -85,B 0,C 180,E1 -18187.662,E2 -18187.662} C_VEL
LIN {X 0,Y 263.37,Z 461.302,A -85,B 0,C 180,E1 -18190.766,E2 -18190.766} C_VEL
LIN {X 0,Y 263.341,Z 461.305,A -85,B 0,C 180,E1 -18195.479,E2 -18195.479} C_VEL
LIN {X 0,Y 263.261,Z 461.317,A -85,B 0,C 180,E1 -18200.307,E2 -18200.307} C_VEL
LIN {X 0,Y 263.206,Z 461.321,A -85,B 0,C 180,E1 -18205.292,E2 -18205.292} C_VEL
LIN {X 0,Y 263.177,Z 461.325,A -85,B 0,C 180,E1 -18208.73,E2 -18208.73} C_VEL
LIN {X 0,Y 263.131,Z 461.335,A -85,B 0,C 180,E1 -18212.289,E2 -18212.289} C_VEL
LIN {X 0,Y 263.174,Z 461.328,A -85,B 0,C 180,E1 -18215.981,E2 -18215.981} C_VEL
LIN {X 0,Y 263.104,Z 461.337,A -85,B 0,C 180,E1 -18219.873,E2 -18219.873} C_VEL
LIN {X 0,Y 263.123,Z 461.335,A -85,B 0,C 180,E1 -18223.985,E2 -18223.985} C_VEL
LIN {X 0,Y 263.155,Z 461.329,A -85,B 0,C 180,E1 -18228.4,E2 -18228.4} C_VEL
LIN {X 0,Y 263.189,Z 461.326,A -85,B 0,C 180,E1 -18232.109,E2 -18232.109} C_VEL
LIN {X 0,Y 263.185,Z 461.327,A -85,B 0,C 180,E1 -18235.891,E2 -18235.891} C_VEL
LIN {X 0,Y 263.155,Z 461.33,A -85,B 0,C 180,E1 -18239.508,E2 -18239.508} C_VEL
LIN {X 0,Y 263.199,Z 461.321,A -85,B 0,C 180,E1 -18243.004,E2 -18243.004} C_VEL
LIN {X 0,Y 263.186,Z 461.324,A -85,B 0,C 180,E1 -18246.388,E2 -18246.388} C_VEL
LIN {X 0,Y 263.266,Z 461.318,A -85,B 0,C 180,E1 -18249.694,E2 -18249.694} C_VEL
LIN {X 0,Y 263.354,Z 461.303,A -85,B 0,C 180,E1 -18254.522,E2 -18254.522} C_VEL
LIN {X 0,Y 263.358,Z 461.304,A -85,B 0,C 180,E1 -18259.234,E2 -18259.234} C_VEL
LIN {X 0,Y 263.533,Z 461.28,A -85,B 0,C 180,E1 -18262.337,E2 -18262.337} C_VEL
LIN {X 0,Y 263.754,Z 461.252,A -85,B 0,C 180,E1 -18268.473,E2 -18268.473} C_VEL
LIN {X 0,Y 263.754,Z 461.256,A -85,B 0,C 180,E1 -18271.527,E2 -18271.527} C_VEL
LIN {X 0,Y 263.561,Z 461.277,A -85,B 0,C 180,E1 -18277.662,E2 -18277.662} C_VEL
LIN {X 0,Y 263.358,Z 461.302,A -85,B 0,C 180,E1 -18280.766,E2 -18280.766} C_VEL
LIN {X 0,Y 263.354,Z 461.306,A -85,B 0,C 180,E1 -18285.478,E2 -18285.478} C_VEL
LIN {X 0,Y 263.266,Z 461.315,A -85,B 0,C 180,E1 -18290.306,E2 -18290.306} C_VEL
LIN {X 0,Y 263.211,Z 461.324,A -85,B 0,C 180,E1 -18295.291,E2 -18295.291} C_VEL
LIN {X 0,Y 263.181,Z 461.328,A -85,B 0,C 180,E1 -18298.729,E2 -18298.729} C_VEL
LIN {X 0,Y 263.099,Z 461.336,A -85,B 0,C 180,E1 -18302.292,E2 -18302.292} C_VEL
LIN {X 0,Y 262.874,Z 461.364,A -85,B 0,C 180,E1 -18306.027,E2 -18306.027} C_VEL
LIN {X 0,Y 262.424,Z 461.424,A -85,B 0,C 180,E1 -18309.996,E2 -18309.996} C_VEL
LIN {X 0,Y 262.226,Z 461.448,A -85,B 0,C 180,E1 -18312.018,E2 -18312.018} C_VEL
LIN {X 0,Y 266.968,Z 477.377,A -85,B 0,C 180,E1 -18313.408,E2 -18313.408} C_VEL
LIN {X 0,Y 270.391,Z 490.913,A -85,B 0,C 180,E1 -18314.786,E2 -18314.786} C_VEL
LIN {X 0,Y 273.368,Z 504.058,A -85,B 0,C 180,E1 -18316.362,E2 -18316.362} C_VEL
LIN {X 0,Y 273.202,Z 508.16,A -85,B 0,C 180,E1 -18316.836,E2 -18316.836} C_VEL
LIN {X 0,Y 271.365,Z 520.609,A -85,B 0,C 180,E1 -18318.409,E2 -18318.409} C_VEL
LIN {X 0,Y 269.415,Z 532.603,A -85,B 0,C 180,E1 -18320.274,E2 -18320.274} C_VEL
LIN {X 0,Y 267.496,Z 544.18,A -85,B 0,C 180,E1 -18322.479,E2 -18322.479} C_VEL
LIN {X 0,Y 265.71,Z 554.428,A -85,B 0,C 180,E1 -18324.858,E2 -18324.858} C_VEL
LIN {X 0,Y 264.193,Z 563.405,A -85,B 0,C 180,E1 -18327.405,E2 -18327.405} C_VEL
LIN {X 0,Y 263.09,Z 570.669,A -85,B 0,C 180,E1 -18329.942,E2 -18329.942} C_VEL
LIN {X 0,Y 262.361,Z 575.794,A -85,B 0,C 180,E1 -18332.125,E2 -18332.125} C_VEL
LIN {X 0,Y 261.792,Z 580.486,A -85,B 0,C 180,E1 -18334.562,E2 -18334.562} C_VEL
LIN {X 0,Y 261.364,Z 584.256,A -85,B 0,C 180,E1 -18337.051,E2 -18337.051} C_VEL
LIN {X 0,Y 261.111,Z 587.771,A -85,B 0,C 180,E1 -18340.396,E2 -18340.396} C_VEL
LIN {X 0,Y 261.139,Z 589.301,A -85,B 0,C 180,E1 -18342.78,E2 -18342.78} C_VEL
LIN {X 0,Y 261.556,Z 590.075,A -85,B 0,C 180,E1 -18346.005,E2 -18346.005} C_VEL
LIN {X 0,Y 262.246,Z 589.443,A -85,B 0,C 180,E1 -18349.187,E2 -18349.187} C_VEL
LIN {X 0,Y 263.504,Z 587.434,A -85,B 0,C 180,E1 -18352.336,E2 -18352.336} C_VEL
LIN {X 0,Y 265.198,Z 584.071,A -85,B 0,C 180,E1 -18355.44,E2 -18355.44} C_VEL
LIN {X 0,Y 267.586,Z 579.209,A -85,B 0,C 180,E1 -18358.495,E2 -18358.495} C_VEL
LIN {X 0,Y 270.53,Z 572.789,A -85,B 0,C 180,E1 -18361.488,E2 -18361.488} C_VEL
LIN {X 0,Y 273.661,Z 565.721,A -85,B 0,C 180,E1 -18364.05,E2 -18364.05} C_VEL
LIN {X 0,Y 277.358,Z 557.069,A -85,B 0,C 180,E1 -18366.547,E2 -18366.547} C_VEL
LIN {X 0,Y 280.947,Z 548.185,A -85,B 0,C 180,E1 -18368.632,E2 -18368.632} C_VEL
LIN {X 0,Y 284.856,Z 537.594,A -85,B 0,C 180,E1 -18370.663,E2 -18370.663} C_VEL
LIN {X 0,Y 288.754,Z 526.027,A -85,B 0,C 180,E1 -18372.475,E2 -18372.475} C_VEL
LIN {X 0,Y 289.472,Z 523.652,A -85,B 0,C 180,E1 -18372.8,E2 -18372.8} C_VEL
LIN {X 0,Y 289.218,Z 520.058,A -85,B 0,C 180,E1 -18373.595,E2 -18373.595} C_VEL
LIN {X 0,Y 287.295,Z 511.211,A -85,B 0,C 180,E1 -18375.811,E2 -18375.811} C_VEL
LIN {X 0,Y 284.295,Z 502.593,A -85,B 0,C 180,E1 -18378.304,E2 -18378.304} C_VEL
LIN {X 0,Y 283.633,Z 500.977,A -85,B 0,C 180,E1 -18378.821,E2 -18378.821} C_VEL
LIN {X 0,Y 281.957,Z 498.594,A -85,B 0,C 180,E1 -18379.859,E2 -18379.859} C_VEL
LIN {X 0,Y 279.865,Z 497.148,A -85,B 0,C 180,E1 -18380.953,E2 -18380.953} C_VEL
LIN {X 0,Y 274.226,Z 494.917,A -85,B 0,C 180,E1 -18384.031,E2 -18384.031} C_VEL
LIN {X 0,Y 273.181,Z 494.067,A -85,B 0,C 180,E1 -18384.825,E2 -18384.825} C_VEL
LIN {X 0,Y 271.466,Z 491.249,A -85,B 0,C 180,E1 -18386.719,E2 -18386.719} C_VEL
LIN {X 0,Y 268.685,Z 488.451,A -85,B 0,C 180,E1 -18390.326,E2 -18390.326} C_VEL
LIN {X 0,Y 268.254,Z 487.412,A -85,B 0,C 180,E1 -18391.599,E2 -18391.599} C_VEL
LIN {X 0,Y 267.531,Z 487.251,A -85,B 0,C 180,E1 -18393.481,E2 -18393.481} C_VEL
LIN {X 0,Y 267.169,Z 487.669,A -85,B 0,C 180,E1 -18395.368,E2 -18395.368} C_VEL
LIN {X 0,Y 267.845,Z 489.466,A -85,B 0,C 180,E1 -18399.03,E2 -18399.03} C_VEL
LIN {X 0,Y 268.699,Z 491.084,A -85,B 0,C 180,E1 -18400.835,E2 -18400.835} C_VEL
LIN {X 0,Y 269.915,Z 495.067,A -85,B 0,C 180,E1 -18403.193,E2 -18403.193} C_VEL
LIN {X 0,Y 271.952,Z 498.588,A -85,B 0,C 180,E1 -18405.382,E2 -18405.382} C_VEL
LIN {X 0,Y 273.265,Z 502.711,A -85,B 0,C 180,E1 -18406.994,E2 -18406.994} C_VEL
LIN {X 0,Y 273.767,Z 503.632,A -85,B 0,C 180,E1 -18407.411,E2 -18407.411} C_VEL
LIN {X 0,Y 275.493,Z 509.616,A -85,B 0,C 180,E1 -18409.326,E2 -18409.326} C_VEL
LIN {X 0,Y 277.18,Z 518.019,A -85,B 0,C 180,E1 -18411.5,E2 -18411.5} C_VEL
LIN {X 0,Y 278.312,Z 526.375,A -85,B 0,C 180,E1 -18413.393,E2 -18413.393} C_VEL
LIN {X 0,Y 278.845,Z 536.234,A -85,B 0,C 180,E1 -18415.435,E2 -18415.435} C_VEL
LIN {X 0,Y 278.409,Z 547.292,A -85,B 0,C 180,E1 -18417.592,E2 -18417.592} C_VEL
LIN {X 0,Y 276.996,Z 556.389,A -85,B 0,C 180,E1 -18419.296,E2 -18419.296} C_VEL
LIN {X 0,Y 275.459,Z 561.299,A -85,B 0,C 180,E1 -18420.165,E2 -18420.165} C_VEL
LIN {X 0,Y 271.193,Z 572.068,A -85,B 0,C 180,E1 -18422.195,E2 -18422.195} C_VEL
LIN {X 0,Y 267.531,Z 581.233,A -85,B 0,C 180,E1 -18424.314,E2 -18424.314} C_VEL
LIN {X 0,Y 263.83,Z 590.264,A -85,B 0,C 180,E1 -18426.864,E2 -18426.864} C_VEL
LIN {X 0,Y 260.715,Z 597.857,A -85,B 0,C 180,E1 -18429.486,E2 -18429.486} C_VEL
LIN {X 0,Y 257.964,Z 604.887,A -85,B 0,C 180,E1 -18432.562,E2 -18432.562} C_VEL
LIN {X 0,Y 256.058,Z 610.39,A -85,B 0,C 180,E1 -18435.699,E2 -18435.699} C_VEL
LIN {X 0,Y 254.773,Z 614.485,A -85,B 0,C 180,E1 -18438.867,E2 -18438.867} C_VEL
LIN {X 0,Y 254.177,Z 617.234,A -85,B 0,C 180,E1 -18442.054,E2 -18442.054} C_VEL
LIN {X 0,Y 254.091,Z 618.665,A -85,B 0,C 180,E1 -18445.24,E2 -18445.24} C_VEL
LIN {X 0,Y 254.203,Z 618.878,A -85,B 0,C 180,E1 -18446.83,E2 -18446.83} C_VEL
LIN {X 0,Y 254.467,Z 618.268,A -85,B 0,C 180,E1 -18450,E2 -18450} C_VEL
LIN {X 0,Y 254.28,Z 616.192,A -85,B 0,C 180,E1 -18453.169,E2 -18453.169} C_VEL
LIN {X 0,Y 254.371,Z 613.148,A -85,B 0,C 180,E1 -18455.936,E2 -18455.936} C_VEL
LIN {X 0,Y 254.473,Z 608.817,A -85,B 0,C 180,E1 -18458.737,E2 -18458.737} C_VEL
LIN {X 0,Y 255.03,Z 602.257,A -85,B 0,C 180,E1 -18461.928,E2 -18461.928} C_VEL
LIN {X 0,Y 255.929,Z 594.902,A -85,B 0,C 180,E1 -18464.715,E2 -18464.715} C_VEL
LIN {X 0,Y 257.384,Z 585.749,A -85,B 0,C 180,E1 -18467.479,E2 -18467.479} C_VEL
LIN {X 0,Y 259.01,Z 576.21,A -85,B 0,C 180,E1 -18469.826,E2 -18469.826} C_VEL
LIN {X 0,Y 261.097,Z 564.707,A -85,B 0,C 180,E1 -18472.138,E2 -18472.138} C_VEL
LIN {X 0,Y 263.175,Z 553.133,A -85,B 0,C 180,E1 -18474.032,E2 -18474.032} C_VEL
LIN {X 0,Y 264.092,Z 546.982,A -85,B 0,C 180,E1 -18474.902,E2 -18474.902} C_VEL
LIN {X 0,Y 263.028,Z 534.324,A -85,B 0,C 180,E1 -18476.586,E2 -18476.586} C_VEL
LIN {X 0,Y 261.18,Z 519.284,A -85,B 0,C 180,E1 -18478.258,E2 -18478.258} C_VEL
LIN {X 0,Y 259.098,Z 504.675,A -85,B 0,C 180,E1 -18479.586,E2 -18479.586} C_VEL
LIN {X 0,Y 256.509,Z 489.06,A -85,B 0,C 180,E1 -18480.744,E2 -18480.744} C_VEL
LIN {X 0,Y 257.559,Z 483.482,A -85,B 0,C 180,E1 -18485.055,E2 -18485.055} C_VEL
LIN {X 0,Y 258.448,Z 478.858,A -85,B 0,C 180,E1 -18488.714,E2 -18488.714} C_VEL
LIN {X 0,Y 258.445,Z 475.264,A -85,B 0,C 180,E1 -18491.7,E2 -18491.7} C_VEL
LIN {X 0,Y 257.61,Z 470.296,A -85,B 0,C 180,E1 -18496.06,E2 -18496.06} C_VEL
LIN {X 0,Y 256.652,Z 465.064,A -85,B 0,C 180,E1 -18500.964,E2 -18500.964} C_VEL
LIN {X 0,Y 256.168,Z 462.204,A -85,B 0,C 180,E1 -18503.853,E2 -18503.853} C_VEL
LIN {X 0,Y 256.09,Z 462.21,A -85,B 0,C 180,E1 -18508.572,E2 -18508.572} C_VEL
LIN {X 0,Y 256.138,Z 462.202,A -85,B 0,C 180,E1 -18512.196,E2 -18512.196} C_VEL
LIN {X 0,Y 256.163,Z 462.197,A -85,B 0,C 180,E1 -18515.699,E2 -18515.699} C_VEL
LIN {X 0,Y 256.163,Z 462.202,A -85,B 0,C 180,E1 -18519.105,E2 -18519.105} C_VEL
LIN {X 0,Y 256.296,Z 462.181,A -85,B 0,C 180,E1 -18524.085,E2 -18524.085} C_VEL
LIN {X 0,Y 256.306,Z 462.184,A -85,B 0,C 180,E1 -18528.934,E2 -18528.934} C_VEL
LIN {X 0,Y 256.536,Z 462.152,A -85,B 0,C 180,E1 -18532.127,E2 -18532.127} C_VEL
LIN {X 0,Y 256.711,Z 462.134,A -85,B 0,C 180,E1 -18538.432,E2 -18538.432} C_VEL
LIN {X 0,Y 256.713,Z 462.128,A -85,B 0,C 180,E1 -18541.569,E2 -18541.569} C_VEL
LIN {X 0,Y 256.537,Z 462.153,A -85,B 0,C 180,E1 -18547.873,E2 -18547.873} C_VEL
LIN {X 0,Y 256.306,Z 462.18,A -85,B 0,C 180,E1 -18551.067,E2 -18551.067} C_VEL
LIN {X 0,Y 256.291,Z 462.184,A -85,B 0,C 180,E1 -18555.916,E2 -18555.916} C_VEL
LIN {X 0,Y 256.164,Z 462.199,A -85,B 0,C 180,E1 -18560.896,E2 -18560.896} C_VEL
LIN {X 0,Y 256.186,Z 462.196,A -85,B 0,C 180,E1 -18565.139,E2 -18565.139} C_VEL
LIN {X 0,Y 256.112,Z 462.204,A -85,B 0,C 180,E1 -18569.6,E2 -18569.6} C_VEL
LIN {X 0,Y 256.075,Z 462.21,A -85,B 0,C 180,E1 -18573.292,E2 -18573.292} C_VEL
LIN {X 0,Y 256.12,Z 462.202,A -85,B 0,C 180,E1 -18577.274,E2 -18577.274} C_VEL
LIN {X 0,Y 256.071,Z 462.213,A -85,B 0,C 180,E1 -18582.182,E2 -18582.182} C_VEL
LIN {X 0,Y 256.07,Z 462.209,A -85,B 0,C 180,E1 -18586.676,E2 -18586.676} C_VEL
LIN {X 0,Y 256.1,Z 462.207,A -85,B 0,C 180,E1 -18590.864,E2 -18590.864} C_VEL
LIN {X 0,Y 256.122,Z 462.202,A -85,B 0,C 180,E1 -18594.814,E2 -18594.814} C_VEL
LIN {X 0,Y 256.094,Z 462.208,A -85,B 0,C 180,E1 -18598.573,E2 -18598.573} C_VEL
LIN {X 0,Y 256.147,Z 462.2,A -85,B 0,C 180,E1 -18602.197,E2 -18602.197} C_VEL
LIN {X 0,Y 256.17,Z 462.201,A -85,B 0,C 180,E1 -18605.7,E2 -18605.7} C_VEL
LIN {X 0,Y 256.169,Z 462.199,A -85,B 0,C 180,E1 -18609.106,E2 -18609.106} C_VEL
LIN {X 0,Y 256.303,Z 462.182,A -85,B 0,C 180,E1 -18614.086,E2 -18614.086} C_VEL
LIN {X 0,Y 256.298,Z 462.185,A -85,B 0,C 180,E1 -18617.328,E2 -18617.328} C_VEL
LIN {X 0,Y 256.496,Z 462.157,A -85,B 0,C 180,E1 -18622.126,E2 -18622.126} C_VEL
LIN {X 0,Y 256.5,Z 462.158,A -85,B 0,C 180,E1 -18626.859,E2 -18626.859} C_VEL
LIN {X 0,Y 256.769,Z 462.122,A -85,B 0,C 180,E1 -18630,E2 -18630} C_VEL
LIN {X 0,Y 256.502,Z 462.159,A -85,B 0,C 180,E1 -18633.141,E2 -18633.141} C_VEL
LIN {X 0,Y 256.518,Z 462.153,A -85,B 0,C 180,E1 -18637.873,E2 -18637.873} C_VEL
LIN {X 0,Y 256.298,Z 462.183,A -85,B 0,C 180,E1 -18642.672,E2 -18642.672} C_VEL
LIN {X 0,Y 256.286,Z 462.184,A -85,B 0,C 180,E1 -18646.302,E2 -18646.302} C_VEL
LIN {X 0,Y 256.16,Z 462.204,A -85,B 0,C 180,E1 -18651.119,E2 -18651.119} C_VEL
LIN {X 0,Y 256.191,Z 462.199,A -85,B 0,C 180,E1 -18655.138,E2 -18655.138} C_VEL
LIN {X 0,Y 256.114,Z 462.207,A -85,B 0,C 180,E1 -18659.599,E2 -18659.599} C_VEL
LIN {X 0,Y 255.99,Z 462.223,A -85,B 0,C 180,E1 -18663.303,E2 -18663.303} C_VEL
LIN {X 0,Y 255.693,Z 462.26,A -85,B 0,C 180,E1 -18667.206,E2 -18667.206} C_VEL
LIN {X 0,Y 255.247,Z 462.316,A -85,B 0,C 180,E1 -18671.477,E2 -18671.477} C_VEL
LIN {X 0,Y 259.302,Z 475.489,A -85,B 0,C 180,E1 -18672.655,E2 -18672.655} C_VEL
LIN {X 0,Y 262.843,Z 488.924,A -85,B 0,C 180,E1 -18674.042,E2 -18674.042} C_VEL
LIN {X 0,Y 266.069,Z 503.245,A -85,B 0,C 180,E1 -18675.765,E2 -18675.765} C_VEL
LIN {X 0,Y 266.599,Z 506.922,A -85,B 0,C 180,E1 -18676.248,E2 -18676.248} C_VEL
LIN {X 0,Y 264.738,Z 519.332,A -85,B 0,C 180,E1 -18677.811,E2 -18677.811} C_VEL
LIN {X 0,Y 262.658,Z 532.1,A -85,B 0,C 180,E1 -18679.795,E2 -18679.795} C_VEL
LIN {X 0,Y 260.737,Z 543.263,A -85,B 0,C 180,E1 -18681.933,E2 -18681.933} C_VEL
LIN {X 0,Y 259.117,Z 552.56,A -85,B 0,C 180,E1 -18684.074,E2 -18684.074} C_VEL
LIN {X 0,Y 257.541,Z 561.182,A -85,B 0,C 180,E1 -18686.454,E2 -18686.454} C_VEL
LIN {X 0,Y 256.303,Z 568.934,A -85,B 0,C 180,E1 -18689.06,E2 -18689.06} C_VEL
LIN {X 0,Y 255.403,Z 575.331,A -85,B 0,C 180,E1 -18691.707,E2 -18691.707} C_VEL
LIN {X 0,Y 254.662,Z 580.981,A -85,B 0,C 180,E1 -18694.674,E2 -18694.674} C_VEL
LIN {X 0,Y 254.247,Z 584.729,A -85,B 0,C 180,E1 -18697.232,E2 -18697.232} C_VEL
LIN {X 0,Y 254.031,Z 588.195,A -85,B 0,C 180,E1 -18700.61,E2 -18700.61} C_VEL
LIN {X 0,Y 254.143,Z 590.109,A -85,B 0,C 180,E1 -18703.946,E2 -18703.946} C_VEL
LIN {X 0,Y 254.432,Z 590.511,A -85,B 0,C 180,E1 -18705.605,E2 -18705.605} C_VEL
LIN {X 0,Y 255.085,Z 590.255,A -85,B 0,C 180,E1 -18708.88,E2 -18708.88} C_VEL
LIN {X 0,Y 256.324,Z 588.596,A -85,B 0,C 180,E1 -18712.12,E2 -18712.12} C_VEL
LIN {X 0,Y 258.042,Z 585.569,A -85,B 0,C 180,E1 -18715.313,E2 -18715.313} C_VEL
LIN {X 0,Y 260.452,Z 581.136,A -85,B 0,C 180,E1 -18718.453,E2 -18718.453} C_VEL
LIN {X 0,Y 263.476,Z 575.183,A -85,B 0,C 180,E1 -18721.528,E2 -18721.528} C_VEL
LIN {X 0,Y 267.175,Z 567.555,A -85,B 0,C 180,E1 -18724.526,E2 -18724.526} C_VEL
LIN {X 0,Y 271.011,Z 559.233,A -85,B 0,C 180,E1 -18727.075,E2 -18727.075} C_VEL
LIN {X 0,Y 275.402,Z 549.054,A -85,B 0,C 180,E1 -18729.548,E2 -18729.548} C_VEL
LIN {X 0,Y 279.552,Z 538.654,A -85,B 0,C 180,E1 -18731.602,E2 -18731.602} C_VEL
LIN {X 0,Y 283.637,Z 527.269,A -85,B 0,C 180,E1 -18733.424,E2 -18733.424} C_VEL
LIN {X 0,Y 284.019,Z 526.053,A -85,B 0,C 180,E1 -18733.597,E2 -18733.597} C_VEL
LIN {X 0,Y 283.252,Z 519.863,A -85,B 0,C 180,E1 -18735.168,E2 -18735.168} C_VEL
LIN {X 0,Y 281.77,Z 513.499,A -85,B 0,C 180,E1 -18736.943,E2 -18736.943} C_VEL
LIN {X 0,Y 279.395,Z 506.28,A -85,B 0,C 180,E1 -18739.251,E2 -18739.251} C_VEL
LIN {X 0,Y 276.343,Z 499.276,A -85,B 0,C 180,E1 -18741.977,E2 -18741.977} C_VEL
LIN {X 0,Y 273.865,Z 494.809,A -85,B 0,C 180,E1 -18744.242,E2 -18744.242} C_VEL
LIN {X 0,Y 273.181,Z 494.067,A -85,B 0,C 180,E1 -18744.825,E2 -18744.825} C_VEL
LIN {X 0,Y 271.655,Z 493.261,A -85,B 0,C 180,E1 -18746.013,E2 -18746.013} C_VEL
LIN {X 0,Y 268.827,Z 493.856,A -85,B 0,C 180,E1 -18748.028,E2 -18748.028} C_VEL
LIN {X 0,Y 266.887,Z 494.673,A -85,B 0,C 180,E1 -18749.681,E2 -18749.681} C_VEL
LIN {X 0,Y 265.956,Z 494.661,A -85,B 0,C 180,E1 -18750.947,E2 -18750.947} C_VEL
LIN {X 0,Y 265.792,Z 494.431,A -85,B 0,C 180,E1 -18751.371,E2 -18751.371} C_VEL
LIN {X 0,Y 265.577,Z 493.97,A -85,B 0,C 180,E1 -18752.134,E2 -18752.134} C_VEL
LIN {X 0,Y 264.867,Z 494.204,A -85,B 0,C 180,E1 -18754.66,E2 -18754.66} C_VEL
LIN {X 0,Y 264.957,Z 495.298,A -85,B 0,C 180,E1 -18757.595,E2 -18757.595} C_VEL
LIN {X 0,Y 265.768,Z 496.86,A -85,B 0,C 180,E1 -18759.927,E2 -18759.927} C_VEL
LIN {X 0,Y 267.952,Z 503.199,A -85,B 0,C 180,E1 -18764.098,E2 -18764.098} C_VEL
LIN {X 0,Y 268.731,Z 504.978,A -85,B 0,C 180,E1 -18765.081,E2 -18765.081} C_VEL
LIN {X 0,Y 270.274,Z 509.967,A -85,B 0,C 180,E1 -18767.147,E2 -18767.147} C_VEL
LIN {X 0,Y 271.564,Z 515.635,A -85,B 0,C 180,E1 -18768.972,E2 -18768.972} C_VEL
LIN {X 0,Y 272.919,Z 524.792,A -85,B 0,C 180,E1 -18771.427,E2 -18771.427} C_VEL
LIN {X 0,Y 273.528,Z 534.972,A -85,B 0,C 180,E1 -18773.776,E2 -18773.776} C_VEL
LIN {X 0,Y 273.195,Z 545.259,A -85,B 0,C 180,E1 -18775.941,E2 -18775.941} C_VEL
LIN {X 0,Y 272.132,Z 553.389,A -85,B 0,C 180,E1 -18777.597,E2 -18777.597} C_VEL
LIN {X 0,Y 270.472,Z 560.445,A -85,B 0,C 180,E1 -18778.982,E2 -18778.982} C_VEL
LIN {X 0,Y 266.045,Z 570.994,A -85,B 0,C 180,E1 -18780.982,E2 -18780.982} C_VEL
LIN {X 0,Y 261.787,Z 580.787,A -85,B 0,C 180,E1 -18783.278,E2 -18783.278} C_VEL
LIN {X 0,Y 257.851,Z 589.815,A -85,B 0,C 180,E1 -18785.868,E2 -18785.868} C_VEL
LIN {X 0,Y 254.948,Z 596.296,A -85,B 0,C 180,E1 -18788.152,E2 -18788.152} C_VEL
LIN {X 0,Y 251.812,Z 603.539,A -85,B 0,C 180,E1 -18791.28,E2 -18791.28} C_VEL
LIN {X 0,Y 249.575,Z 609.236,A -85,B 0,C 180,E1 -18794.484,E2 -18794.484} C_VEL
LIN {X 0,Y 248.319,Z 612.529,A -85,B 0,C 180,E1 -18796.914,E2 -18796.914} C_VEL
LIN {X 0,Y 247.359,Z 615.807,A -85,B 0,C 180,E1 -18800.185,E2 -18800.185} C_VEL
LIN {X 0,Y 246.998,Z 617.765,A -85,B 0,C 180,E1 -18803.465,E2 -18803.465} C_VEL
LIN {X 0,Y 247.129,Z 618.405,A -85,B 0,C 180,E1 -18806.739,E2 -18806.739} C_VEL
LIN {X 0,Y 247.386,Z 617.672,A -85,B 0,C 180,E1 -18810,E2 -18810} C_VEL
LIN {X 0,Y 247.216,Z 615.47,A -85,B 0,C 180,E1 -18813.259,E2 -18813.259} C_VEL
LIN {X 0,Y 247.316,Z 612.5,A -85,B 0,C 180,E1 -18815.959,E2 -18815.959} C_VEL
LIN {X 0,Y 247.417,Z 607.861,A -85,B 0,C 180,E1 -18818.988,E2 -18818.988} C_VEL
LIN {X 0,Y 247.835,Z 602.999,A -85,B 0,C 180,E1 -18821.449,E2 -18821.449} C_VEL
LIN {X 0,Y 248.705,Z 595.935,A -85,B 0,C 180,E1 -18824.315,E2 -18824.315} C_VEL
LIN {X 0,Y 249.958,Z 587.493,A -85,B 0,C 180,E1 -18827.066,E2 -18827.066} C_VEL
LIN {X 0,Y 251.671,Z 578.023,A -85,B 0,C 180,E1 -18829.578,E2 -18829.578} C_VEL
LIN {X 0,Y 253.643,Z 566.966,A -85,B 0,C 180,E1 -18831.966,E2 -18831.966} C_VEL
LIN {X 0,Y 255.455,Z 557.125,A -85,B 0,C 180,E1 -18833.725,E2 -18833.725} C_VEL
LIN {X 0,Y 257.077,Z 548.119,A -85,B 0,C 180,E1 -18835.08,E2 -18835.08} C_VEL
LIN {X 0,Y 256.251,Z 536.711,A -85,B 0,C 180,E1 -18836.686,E2 -18836.686} C_VEL
LIN {X 0,Y 254.734,Z 523.251,A -85,B 0,C 180,E1 -18838.313,E2 -18838.313} C_VEL
LIN {X 0,Y 252.79,Z 508.602,A -85,B 0,C 180,E1 -18839.782,E2 -18839.782} C_VEL
LIN {X 0,Y 250.266,Z 493.09,A -85,B 0,C 180,E1 -18841.006,E2 -18841.006} C_VEL
LIN {X 0,Y 249.543,Z 488.71,A -85,B 0,C 180,E1 -18841.32,E2 -18841.32} C_VEL
LIN {X 0,Y 250.751,Z 482.807,A -85,B 0,C 180,E1 -18846.056,E2 -18846.056} C_VEL
LIN {X 0,Y 251.31,Z 479.866,A -85,B 0,C 180,E1 -18848.461,E2 -18848.461} C_VEL
LIN {X 0,Y 251.449,Z 476.849,A -85,B 0,C 180,E1 -18851.005,E2 -18851.005} C_VEL
LIN {X 0,Y 250.878,Z 472.974,A -85,B 0,C 180,E1 -18854.453,E2 -18854.453} C_VEL
LIN {X 0,Y 250.247,Z 469.561,A -85,B 0,C 180,E1 -18857.622,E2 -18857.622} C_VEL
LIN {X 0,Y 249.461,Z 465.017,A -85,B 0,C 180,E1 -18862.076,E2 -18862.076} C_VEL
LIN {X 0,Y 249.123,Z 463.082,A -85,B 0,C 180,E1 -18864.193,E2 -18864.193} C_VEL
LIN {X 0,Y 249.037,Z 463.087,A -85,B 0,C 180,E1 -18867.844,E2 -18867.844} C_VEL
LIN {X 0,Y 249.094,Z 463.081,A -85,B 0,C 180,E1 -18871.338,E2 -18871.338} C_VEL
LIN {X 0,Y 249.148,Z 463.073,A -85,B 0,C 180,E1 -18874.968,E2 -18874.968} C_VEL
LIN {X 0,Y 249.107,Z 463.078,A -85,B 0,C 180,E1 -18880.211,E2 -18880.211} C_VEL
LIN {X 0,Y 249.239,Z 463.059,A -85,B 0,C 180,E1 -18883.622,E2 -18883.622} C_VEL
LIN {X 0,Y 249.249,Z 463.064,A -85,B 0,C 180,E1 -18888.617,E2 -18888.617} C_VEL
LIN {X 0,Y 249.477,Z 463.031,A -85,B 0,C 180,E1 -18891.903,E2 -18891.903} C_VEL
LIN {X 0,Y 249.433,Z 463.041,A -85,B 0,C 180,E1 -18896.77,E2 -18896.77} C_VEL
LIN {X 0,Y 249.724,Z 463.001,A -85,B 0,C 180,E1 -18900,E2 -18900} C_VEL
LIN {X 0,Y 249.438,Z 463.036,A -85,B 0,C 180,E1 -18903.231,E2 -18903.231} C_VEL
LIN {X 0,Y 249.479,Z 463.033,A -85,B 0,C 180,E1 -18908.098,E2 -18908.098} C_VEL
LIN {X 0,Y 249.249,Z 463.058,A -85,B 0,C 180,E1 -18911.384,E2 -18911.384} C_VEL
LIN {X 0,Y 249.215,Z 463.067,A -85,B 0,C 180,E1 -18916.504,E2 -18916.504} C_VEL
LIN {X 0,Y 249.085,Z 463.08,A -85,B 0,C 180,E1 -18921.519,E2 -18921.519} C_VEL
LIN {X 0,Y 249.128,Z 463.075,A -85,B 0,C 180,E1 -18925.483,E2 -18925.483} C_VEL
LIN {X 0,Y 249.081,Z 463.079,A -85,B 0,C 180,E1 -18928.994,E2 -18928.994} C_VEL
LIN {X 0,Y 249.031,Z 463.09,A -85,B 0,C 180,E1 -18932.426,E2 -18932.426} C_VEL
LIN {X 0,Y 249.062,Z 463.083,A -85,B 0,C 180,E1 -18936.341,E2 -18936.341} C_VEL
LIN {X 0,Y 249.005,Z 463.092,A -85,B 0,C 180,E1 -18940.479,E2 -18940.479} C_VEL
LIN {X 0,Y 249.004,Z 463.089,A -85,B 0,C 180,E1 -18944.88,E2 -18944.88} C_VEL
LIN {X 0,Y 249.03,Z 463.087,A -85,B 0,C 180,E1 -18947.367,E2 -18947.367} C_VEL
LIN {X 0,Y 249.049,Z 463.087,A -85,B 0,C 180,E1 -18951.624,E2 -18951.624} C_VEL
LIN {X 0,Y 249.063,Z 463.084,A -85,B 0,C 180,E1 -18955.643,E2 -18955.643} C_VEL
LIN {X 0,Y 249.055,Z 463.086,A -85,B 0,C 180,E1 -18959.474,E2 -18959.474} C_VEL
LIN {X 0,Y 249.078,Z 463.08,A -85,B 0,C 180,E1 -18963.163,E2 -18963.163} C_VEL
LIN {X 0,Y 249.082,Z 463.081,A -85,B 0,C 180,E1 -18966.733,E2 -18966.733} C_VEL
LIN {X 0,Y 249.113,Z 463.077,A -85,B 0,C 180,E1 -18970.212,E2 -18970.212} C_VEL
LIN {X 0,Y 249.245,Z 463.063,A -85,B 0,C 180,E1 -18973.622,E2 -18973.622} C_VEL
LIN {X 0,Y 249.248,Z 463.06,A -85,B 0,C 180,E1 -18978.617,E2 -18978.617} C_VEL
LIN {X 0,Y 249.44,Z 463.037,A -85,B 0,C 180,E1 -18981.902,E2 -18981.902} C_VEL
LIN {X 0,Y 249.436,Z 463.037,A -85,B 0,C 180,E1 -18986.77,E2 -18986.77} C_VEL
LIN {X 0,Y 249.732,Z 462.999,A -85,B 0,C 180,E1 -18990,E2 -18990} C_VEL
LIN {X 0,Y 249.439,Z 463.04,A -85,B 0,C 180,E1 -18993.23,E2 -18993.23} C_VEL
LIN {X 0,Y 249.457,Z 463.034,A -85,B 0,C 180,E1 -18996.47,E2 -18996.47} C_VEL
LIN {X 0,Y 249.346,Z 463.047,A -85,B 0,C 180,E1 -18999.736,E2 -18999.736} C_VEL
LIN {X 0,Y 249.209,Z 463.067,A -85,B 0,C 180,E1 -19004.703,E2 -19004.703} C_VEL
LIN {X 0,Y 249.143,Z 463.072,A -85,B 0,C 180,E1 -19008.077,E2 -19008.077} C_VEL
LIN {X 0,Y 249.09,Z 463.082,A -85,B 0,C 180,E1 -19011.517,E2 -19011.517} C_VEL
LIN {X 0,Y 249.133,Z 463.076,A -85,B 0,C 180,E1 -19015.482,E2 -19015.482} C_VEL
LIN {X 0,Y 249.085,Z 463.085,A -85,B 0,C 180,E1 -19018.993,E2 -19018.993} C_VEL
LIN {X 0,Y 248.972,Z 463.096,A -85,B 0,C 180,E1 -19022.434,E2 -19022.434} C_VEL
LIN {X 0,Y 248.714,Z 463.129,A -85,B 0,C 180,E1 -19026.398,E2 -19026.398} C_VEL
LIN {X 0,Y 248.244,Z 463.19,A -85,B 0,C 180,E1 -19030.929,E2 -19030.929} C_VEL
LIN {X 0,Y 252.261,Z 475.859,A -85,B 0,C 180,E1 -19032.106,E2 -19032.106} C_VEL
LIN {X 0,Y 256.095,Z 490.525,A -85,B 0,C 180,E1 -19033.661,E2 -19033.661} C_VEL
LIN {X 0,Y 259.147,Z 504.253,A -85,B 0,C 180,E1 -19035.387,E2 -19035.387} C_VEL
LIN {X 0,Y 259.743,Z 507.255,A -85,B 0,C 180,E1 -19035.807,E2 -19035.807} C_VEL
LIN {X 0,Y 257.74,Z 520.675,A -85,B 0,C 180,E1 -19037.555,E2 -19037.555} C_VEL
LIN {X 0,Y 255.704,Z 532.781,A -85,B 0,C 180,E1 -19039.508,E2 -19039.508} C_VEL
LIN {X 0,Y 253.725,Z 543.886,A -85,B 0,C 180,E1 -19041.7,E2 -19041.7} C_VEL
LIN {X 0,Y 251.876,Z 553.999,A -85,B 0,C 180,E1 -19044.129,E2 -19044.129} C_VEL
LIN {X 0,Y 250.19,Z 563.381,A -85,B 0,C 180,E1 -19046.882,E2 -19046.882} C_VEL
LIN {X 0,Y 249.058,Z 570.574,A -85,B 0,C 180,E1 -19049.473,E2 -19049.473} C_VEL
LIN {X 0,Y 248.168,Z 576.643,A -85,B 0,C 180,E1 -19052.152,E2 -19052.152} C_VEL
LIN {X 0,Y 247.459,Z 582.336,A -85,B 0,C 180,E1 -19055.341,E2 -19055.341} C_VEL
LIN {X 0,Y 247.009,Z 586.236,A -85,B 0,C 180,E1 -19058.291,E2 -19058.291} C_VEL
LIN {X 0,Y 246.945,Z 587.982,A -85,B 0,C 180,E1 -19060.03,E2 -19060.03} C_VEL
LIN {X 0,Y 247.007,Z 590.242,A -85,B 0,C 180,E1 -19063.469,E2 -19063.469} C_VEL
LIN {X 0,Y 247.264,Z 590.816,A -85,B 0,C 180,E1 -19065.178,E2 -19065.178} C_VEL
LIN {X 0,Y 247.902,Z 590.914,A -85,B 0,C 180,E1 -19068.553,E2 -19068.553} C_VEL
LIN {X 0,Y 249.119,Z 589.633,A -85,B 0,C 180,E1 -19071.891,E2 -19071.891} C_VEL
LIN {X 0,Y 250.874,Z 587.021,A -85,B 0,C 180,E1 -19075.179,E2 -19075.179} C_VEL
LIN {X 0,Y 253.284,Z 583.021,A -85,B 0,C 180,E1 -19078.41,E2 -19078.41} C_VEL
LIN {X 0,Y 256.391,Z 577.508,A -85,B 0,C 180,E1 -19081.57,E2 -19081.57} C_VEL
LIN {X 0,Y 260.131,Z 570.39,A -85,B 0,C 180,E1 -19084.649,E2 -19084.649} C_VEL
LIN {X 0,Y 264.1,Z 562.568,A -85,B 0,C 180,E1 -19087.261,E2 -19087.261} C_VEL
LIN {X 0,Y 268.61,Z 553.155,A -85,B 0,C 180,E1 -19089.792,E2 -19089.792} C_VEL
LIN {X 0,Y 272.991,Z 543.07,A -85,B 0,C 180,E1 -19091.966,E2 -19091.966} C_VEL
LIN {X 0,Y 277.815,Z 530.759,A -85,B 0,C 180,E1 -19094.093,E2 -19094.093} C_VEL
LIN {X 0,Y 278.23,Z 529.665,A -85,B 0,C 180,E1 -19094.258,E2 -19094.258} C_VEL
LIN {X 0,Y 278.549,Z 527.933,A -85,B 0,C 180,E1 -19094.614,E2 -19094.614} C_VEL
LIN {X 0,Y 277.494,Z 520.387,A -85,B 0,C 180,E1 -19096.733,E2 -19096.733} C_VEL
LIN {X 0,Y 275.386,Z 512.377,A -85,B 0,C 180,E1 -19099.376,E2 -19099.376} C_VEL
LIN {X 0,Y 272.888,Z 505.831,A -85,B 0,C 180,E1 -19102.008,E2 -19102.008} C_VEL
LIN {X 0,Y 270.487,Z 500.892,A -85,B 0,C 180,E1 -19104.58,E2 -19104.58} C_VEL
LIN {X 0,Y 268.384,Z 497.504,A -85,B 0,C 180,E1 -19107.086,E2 -19107.086} C_VEL
LIN {X 0,Y 265.792,Z 494.431,A -85,B 0,C 180,E1 -19111.371,E2 -19111.371} C_VEL
LIN {X 0,Y 265.436,Z 494.282,A -85,B 0,C 180,E1 -19112.208,E2 -19112.208} C_VEL
LIN {X 0,Y 264.612,Z 495.336,A -85,B 0,C 180,E1 -19113.45,E2 -19113.45} C_VEL
LIN {X 0,Y 262.627,Z 500.243,A -85,B 0,C 180,E1 -19116.289,E2 -19116.289} C_VEL
LIN {X 0,Y 262.328,Z 501.858,A -85,B 0,C 180,E1 -19117.559,E2 -19117.559} C_VEL
LIN {X 0,Y 262.375,Z 502.147,A -85,B 0,C 180,E1 -19117.995,E2 -19117.995} C_VEL
LIN {X 0,Y 262.985,Z 503.572,A -85,B 0,C 180,E1 -19119.894,E2 -19119.894} C_VEL
LIN {X 0,Y 265.078,Z 510.146,A -85,B 0,C 180,E1 -19124.288,E2 -19124.288} C_VEL
LIN {X 0,Y 266.517,Z 515.715,A -85,B 0,C 180,E1 -19126.717,E2 -19126.717} C_VEL
LIN {X 0,Y 267.509,Z 521.49,A -85,B 0,C 180,E1 -19128.651,E2 -19128.651} C_VEL
LIN {X 0,Y 268.272,Z 530.139,A -85,B 0,C 180,E1 -19131.044,E2 -19131.044} C_VEL
LIN {X 0,Y 268.291,Z 540.586,A -85,B 0,C 180,E1 -19133.557,E2 -19133.557} C_VEL
LIN {X 0,Y 267.239,Z 551.17,A -85,B 0,C 180,E1 -19135.893,E2 -19135.893} C_VEL
LIN {X 0,Y 265.575,Z 559.202,A -85,B 0,C 180,E1 -19137.597,E2 -19137.597} C_VEL
LIN {X 0,Y 264.025,Z 563.493,A -85,B 0,C 180,E1 -19138.439,E2 -19138.439} C_VEL
LIN {X 0,Y 258.918,Z 574.639,A -85,B 0,C 180,E1 -19140.753,E2 -19140.753} C_VEL
LIN {X 0,Y 254.931,Z 583.176,A -85,B 0,C 180,E1 -19142.944,E2 -19142.944} C_VEL
LIN {X 0,Y 251.432,Z 590.499,A -85,B 0,C 180,E1 -19145.211,E2 -19145.211} C_VEL
LIN {X 0,Y 248.39,Z 596.857,A -85,B 0,C 180,E1 -19147.545,E2 -19147.545} C_VEL
LIN {X 0,Y 245.087,Z 603.812,A -85,B 0,C 180,E1 -19150.746,E2 -19150.746} C_VEL
LIN {X 0,Y 242.682,Z 609.287,A -85,B 0,C 180,E1 -19154.031,E2 -19154.031} C_VEL
LIN {X 0,Y 241.385,Z 612.49,A -85,B 0,C 180,E1 -19156.531,E2 -19156.531} C_VEL
LIN {X 0,Y 240.329,Z 615.597,A -85,B 0,C 180,E1 -19159.895,E2 -19159.895} C_VEL
LIN {X 0,Y 239.906,Z 617.419,A -85,B 0,C 180,E1 -19163.271,E2 -19163.271} C_VEL
LIN {X 0,Y 240.056,Z 617.928,A -85,B 0,C 180,E1 -19166.643,E2 -19166.643} C_VEL
LIN {X 0,Y 240.304,Z 617.078,A -85,B 0,C 180,E1 -19170,E2 -19170} C_VEL
LIN {X 0,Y 240.153,Z 614.74,A -85,B 0,C 180,E1 -19173.355,E2 -19173.355} C_VEL
LIN {X 0,Y 240.259,Z 611.837,A -85,B 0,C 180,E1 -19175.98,E2 -19175.98} C_VEL
LIN {X 0,Y 240.382,Z 606.861,A -85,B 0,C 180,E1 -19179.253,E2 -19179.253} C_VEL
LIN {X 0,Y 240.835,Z 601.843,A -85,B 0,C 180,E1 -19181.787,E2 -19181.787} C_VEL
LIN {X 0,Y 241.74,Z 594.621,A -85,B 0,C 180,E1 -19184.737,E2 -19184.737} C_VEL
LIN {X 0,Y 242.984,Z 586.704,A -85,B 0,C 180,E1 -19187.354,E2 -19187.354} C_VEL
LIN {X 0,Y 244.589,Z 577.999,A -85,B 0,C 180,E1 -19189.732,E2 -19189.732} C_VEL
LIN {X 0,Y 246.592,Z 567.095,A -85,B 0,C 180,E1 -19192.187,E2 -19192.187} C_VEL
LIN {X 0,Y 248.667,Z 556.174,A -85,B 0,C 180,E1 -19194.192,E2 -19194.192} C_VEL
LIN {X 0,Y 250.139,Z 548.001,A -85,B 0,C 180,E1 -19195.459,E2 -19195.459} C_VEL
LIN {X 0,Y 249.099,Z 535.865,A -85,B 0,C 180,E1 -19197.222,E2 -19197.222} C_VEL
LIN {X 0,Y 247.524,Z 521.228,A -85,B 0,C 180,E1 -19199.011,E2 -19199.011} C_VEL
LIN {X 0,Y 245.407,Z 505.992,A -85,B 0,C 180,E1 -19200.527,E2 -19200.527} C_VEL
LIN {X 0,Y 242.853,Z 490.328,A -85,B 0,C 180,E1 -19201.772,E2 -19201.772} C_VEL
LIN {X 0,Y 242.595,Z 488.298,A -85,B 0,C 180,E1 -19201.974,E2 -19201.974} C_VEL
LIN {X 0,Y 243.695,Z 483.254,A -85,B 0,C 180,E1 -19206.148,E2 -19206.148} C_VEL
LIN {X 0,Y 244.316,Z 479.581,A -85,B 0,C 180,E1 -19209.26,E2 -19209.26} C_VEL
LIN {X 0,Y 244.313,Z 476.945,A -85,B 0,C 180,E1 -19211.589,E2 -19211.589} C_VEL
LIN {X 0,Y 243.718,Z 473.174,A -85,B 0,C 180,E1 -19215.05,E2 -19215.05} C_VEL
LIN {X 0,Y 242.981,Z 469.352,A -85,B 0,C 180,E1 -19218.765,E2 -19218.765} C_VEL
LIN {X 0,Y 242.205,Z 464.71,A -85,B 0,C 180,E1 -19223.5,E2 -19223.5} C_VEL
LIN {X 0,Y 242.074,Z 463.96,A -85,B 0,C 180,E1 -19224.504,E2 -19224.504} C_VEL
LIN {X 0,Y 241.973,Z 463.968,A -85,B 0,C 180,E1 -19228.48,E2 -19228.48} C_VEL
LIN {X 0,Y 242.006,Z 463.963,A -85,B 0,C 180,E1 -19232.313,E2 -19232.313} C_VEL
LIN {X 0,Y 242.054,Z 463.954,A -85,B 0,C 180,E1 -19236.016,E2 -19236.016} C_VEL
LIN {X 0,Y 242.034,Z 463.959,A -85,B 0,C 180,E1 -19239.608,E2 -19239.608} C_VEL
LIN {X 0,Y 242.16,Z 463.942,A -85,B 0,C 180,E1 -19243.278,E2 -19243.278} C_VEL
LIN {X 0,Y 242.183,Z 463.942,A -85,B 0,C 180,E1 -19248.28,E2 -19248.28} C_VEL
LIN {X 0,Y 242.424,Z 463.909,A -85,B 0,C 180,E1 -19251.666,E2 -19251.666} C_VEL
LIN {X 0,Y 242.257,Z 463.933,A -85,B 0,C 180,E1 -19255.007,E2 -19255.007} C_VEL
LIN {X 0,Y 242.633,Z 463.887,A -85,B 0,C 180,E1 -19258.34,E2 -19258.34} C_VEL
LIN {X 0,Y 242.635,Z 463.881,A -85,B 0,C 180,E1 -19261.66,E2 -19261.66} C_VEL
LIN {X 0,Y 242.428,Z 463.913,A -85,B 0,C 180,E1 -19266.705,E2 -19266.705} C_VEL
LIN {X 0,Y 242.311,Z 463.924,A -85,B 0,C 180,E1 -19270.022,E2 -19270.022} C_VEL
LIN {X 0,Y 242.161,Z 463.943,A -85,B 0,C 180,E1 -19275.142,E2 -19275.142} C_VEL
LIN {X 0,Y 242.07,Z 463.954,A -85,B 0,C 180,E1 -19278.625,E2 -19278.625} C_VEL
LIN {X 0,Y 242.01,Z 463.964,A -85,B 0,C 180,E1 -19282.181,E2 -19282.181} C_VEL
LIN {X 0,Y 242.065,Z 463.956,A -85,B 0,C 180,E1 -19285.839,E2 -19285.839} C_VEL
LIN {X 0,Y 242.029,Z 463.958,A -85,B 0,C 180,E1 -19289.581,E2 -19289.581} C_VEL
LIN {X 0,Y 241.987,Z 463.965,A -85,B 0,C 180,E1 -19293.492,E2 -19293.492} C_VEL
LIN {X 0,Y 241.994,Z 463.962,A -85,B 0,C 180,E1 -19297.582,E2 -19297.582} C_VEL
LIN {X 0,Y 241.937,Z 463.975,A -85,B 0,C 180,E1 -19301.923,E2 -19301.923} C_VEL
LIN {X 0,Y 241.943,Z 463.969,A -85,B 0,C 180,E1 -19306.57,E2 -19306.57} C_VEL
LIN {X 0,Y 241.982,Z 463.967,A -85,B 0,C 180,E1 -19310.287,E2 -19310.287} C_VEL
LIN {X 0,Y 242.038,Z 463.956,A -85,B 0,C 180,E1 -19314.498,E2 -19314.498} C_VEL
LIN {X 0,Y 241.978,Z 463.966,A -85,B 0,C 180,E1 -19318.481,E2 -19318.481} C_VEL
LIN {X 0,Y 242.014,Z 463.96,A -85,B 0,C 180,E1 -19322.314,E2 -19322.314} C_VEL
LIN {X 0,Y 242.06,Z 463.958,A -85,B 0,C 180,E1 -19326.017,E2 -19326.017} C_VEL
LIN {X 0,Y 242.041,Z 463.962,A -85,B 0,C 180,E1 -19329.609,E2 -19329.609} C_VEL
LIN {X 0,Y 242.166,Z 463.942,A -85,B 0,C 180,E1 -19333.279,E2 -19333.279} C_VEL
LIN {X 0,Y 242.184,Z 463.94,A -85,B 0,C 180,E1 -19338.28,E2 -19338.28} C_VEL
LIN {X 0,Y 242.389,Z 463.916,A -85,B 0,C 180,E1 -19341.664,E2 -19341.664} C_VEL
LIN {X 0,Y 242.251,Z 463.933,A -85,B 0,C 180,E1 -19345.007,E2 -19345.007} C_VEL
LIN {X 0,Y 242.639,Z 463.882,A -85,B 0,C 180,E1 -19348.34,E2 -19348.34} C_VEL
LIN {X 0,Y 242.64,Z 463.885,A -85,B 0,C 180,E1 -19351.66,E2 -19351.66} C_VEL
LIN {X 0,Y 242.427,Z 463.91,A -85,B 0,C 180,E1 -19356.659,E2 -19356.659} C_VEL
LIN {X 0,Y 242.271,Z 463.927,A -85,B 0,C 180,E1 -19360.023,E2 -19360.023} C_VEL
LIN {X 0,Y 242.17,Z 463.947,A -85,B 0,C 180,E1 -19365.14,E2 -19365.14} C_VEL
LIN {X 0,Y 242.076,Z 463.954,A -85,B 0,C 180,E1 -19368.624,E2 -19368.624} C_VEL
LIN {X 0,Y 242.016,Z 463.961,A -85,B 0,C 180,E1 -19372.179,E2 -19372.179} C_VEL
LIN {X 0,Y 242.069,Z 463.955,A -85,B 0,C 180,E1 -19375.837,E2 -19375.837} C_VEL
LIN {X 0,Y 242.03,Z 463.962,A -85,B 0,C 180,E1 -19379.58,E2 -19379.58} C_VEL
LIN {X 0,Y 241.849,Z 463.983,A -85,B 0,C 180,E1 -19383.513,E2 -19383.513} C_VEL
LIN {X 0,Y 241.756,Z 463.995,A -85,B 0,C 180,E1 -19385.549,E2 -19385.549} C_VEL
LIN {X 0,Y 241.238,Z 464.062,A -85,B 0,C 180,E1 -19390.327,E2 -19390.327} C_VEL
LIN {X 0,Y 245.754,Z 478.144,A -85,B 0,C 180,E1 -19391.728,E2 -19391.728} C_VEL
LIN {X 0,Y 249.478,Z 492.691,A -85,B 0,C 180,E1 -19393.366,E2 -19393.366} C_VEL
LIN {X 0,Y 252.424,Z 506.22,A -85,B 0,C 180,E1 -19395.15,E2 -19395.15} C_VEL
LIN {X 0,Y 252.769,Z 509.097,A -85,B 0,C 180,E1 -19395.546,E2 -19395.546} C_VEL
LIN {X 0,Y 250.733,Z 521.883,A -85,B 0,C 180,E1 -19397.292,E2 -19397.292} C_VEL
LIN {X 0,Y 248.519,Z 534.465,A -85,B 0,C 180,E1 -19399.426,E2 -19399.426} C_VEL
LIN {X 0,Y 246.555,Z 545.366,A -85,B 0,C 180,E1 -19401.685,E2 -19401.685} C_VEL
LIN {X 0,Y 244.815,Z 554.461,A -85,B 0,C 180,E1 -19403.949,E2 -19403.949} C_VEL
LIN {X 0,Y 243.152,Z 563.57,A -85,B 0,C 180,E1 -19406.689,E2 -19406.689} C_VEL
LIN {X 0,Y 241.938,Z 571.039,A -85,B 0,C 180,E1 -19409.445,E2 -19409.445} C_VEL
LIN {X 0,Y 241.062,Z 577.094,A -85,B 0,C 180,E1 -19412.194,E2 -19412.194} C_VEL
LIN {X 0,Y 240.41,Z 582.024,A -85,B 0,C 180,E1 -19414.988,E2 -19414.988} C_VEL
LIN {X 0,Y 240.002,Z 585.65,A -85,B 0,C 180,E1 -19417.624,E2 -19417.624} C_VEL
LIN {X 0,Y 239.821,Z 589.112,A -85,B 0,C 180,E1 -19421.194,E2 -19421.194} C_VEL
LIN {X 0,Y 240.084,Z 591.045,A -85,B 0,C 180,E1 -19424.724,E2 -19424.724} C_VEL
LIN {X 0,Y 240.725,Z 591.537,A -85,B 0,C 180,E1 -19428.207,E2 -19428.207} C_VEL
LIN {X 0,Y 241.92,Z 590.643,A -85,B 0,C 180,E1 -19431.648,E2 -19431.648} C_VEL
LIN {X 0,Y 243.692,Z 588.39,A -85,B 0,C 180,E1 -19435.036,E2 -19435.036} C_VEL
LIN {X 0,Y 246.125,Z 584.764,A -85,B 0,C 180,E1 -19438.363,E2 -19438.363} C_VEL
LIN {X 0,Y 249.313,Z 579.711,A -85,B 0,C 180,E1 -19441.615,E2 -19441.615} C_VEL
LIN {X 0,Y 253.129,Z 573.099,A -85,B 0,C 180,E1 -19444.778,E2 -19444.778} C_VEL
LIN {X 0,Y 257.164,Z 565.889,A -85,B 0,C 180,E1 -19447.458,E2 -19447.458} C_VEL
LIN {X 0,Y 261.78,Z 557.051,A -85,B 0,C 180,E1 -19450.05,E2 -19450.05} C_VEL
LIN {X 0,Y 266.824,Z 546.433,A -85,B 0,C 180,E1 -19452.53,E2 -19452.53} C_VEL
LIN {X 0,Y 271.633,Z 535.303,A -85,B 0,C 180,E1 -19454.609,E2 -19454.609} C_VEL
LIN {X 0,Y 273.125,Z 531.257,A -85,B 0,C 180,E1 -19455.293,E2 -19455.293} C_VEL
LIN {X 0,Y 272.454,Z 524.446,A -85,B 0,C 180,E1 -19457.368,E2 -19457.368} C_VEL
LIN {X 0,Y 270.641,Z 516.568,A -85,B 0,C 180,E1 -19460.164,E2 -19460.164} C_VEL
LIN {X 0,Y 268.961,Z 511.511,A -85,B 0,C 180,E1 -19462.347,E2 -19462.347} C_VEL
LIN {X 0,Y 266.932,Z 506.858,A -85,B 0,C 180,E1 -19464.914,E2 -19464.914} C_VEL
LIN {X 0,Y 265.501,Z 504.588,A -85,B 0,C 180,E1 -19466.744,E2 -19466.744} C_VEL
LIN {X 0,Y 264.214,Z 502.826,A -85,B 0,C 180,E1 -19468.625,E2 -19468.625} C_VEL
LIN {X 0,Y 262.795,Z 500.513,A -85,B 0,C 180,E1 -19472.335,E2 -19472.335} C_VEL
LIN {X 0,Y 262.277,Z 500.701,A -85,B 0,C 180,E1 -19474.244,E2 -19474.244} C_VEL
LIN {X 0,Y 262.375,Z 502.147,A -85,B 0,C 180,E1 -19477.995,E2 -19477.995} C_VEL
LIN {X 0,Y 262.533,Z 502.945,A -85,B 0,C 180,E1 -19478.831,E2 -19478.831} C_VEL
LIN {X 0,Y 262.431,Z 504.368,A -85,B 0,C 180,E1 -19479.629,E2 -19479.629} C_VEL
LIN {X 0,Y 261.94,Z 508.34,A -85,B 0,C 180,E1 -19481.126,E2 -19481.126} C_VEL
LIN {X 0,Y 261.351,Z 514.905,A -85,B 0,C 180,E1 -19483.361,E2 -19483.361} C_VEL
LIN {X 0,Y 261.605,Z 516.616,A -85,B 0,C 180,E1 -19484.159,E2 -19484.159} C_VEL
LIN {X 0,Y 262.575,Z 521.294,A -85,B 0,C 180,E1 -19486.275,E2 -19486.275} C_VEL
LIN {X 0,Y 263.166,Z 526.553,A -85,B 0,C 180,E1 -19488.116,E2 -19488.116} C_VEL
LIN {X 0,Y 263.428,Z 535.478,A -85,B 0,C 180,E1 -19490.686,E2 -19490.686} C_VEL
LIN {X 0,Y 262.954,Z 544.767,A -85,B 0,C 180,E1 -19493.034,E2 -19493.034} C_VEL
LIN {X 0,Y 261.528,Z 554.497,A -85,B 0,C 180,E1 -19495.298,E2 -19495.298} C_VEL
LIN {X 0,Y 259.233,Z 562.882,A -85,B 0,C 180,E1 -19497.166,E2 -19497.166} C_VEL
LIN {X 0,Y 254.335,Z 573.059,A -85,B 0,C 180,E1 -19499.286,E2 -19499.286} C_VEL
LIN {X 0,Y 249.335,Z 582.89,A -85,B 0,C 180,E1 -19501.828,E2 -19501.828} C_VEL
LIN {X 0,Y 245.63,Z 590.175,A -85,B 0,C 180,E1 -19504.13,E2 -19504.13} C_VEL
LIN {X 0,Y 241.87,Z 597.354,A -85,B 0,C 180,E1 -19506.905,E2 -19506.905} C_VEL
LIN {X 0,Y 238.389,Z 604.085,A -85,B 0,C 180,E1 -19510.182,E2 -19510.182} C_VEL
LIN {X 0,Y 235.817,Z 609.35,A -85,B 0,C 180,E1 -19513.553,E2 -19513.553} C_VEL
LIN {X 0,Y 234.46,Z 612.446,A -85,B 0,C 180,E1 -19516.125,E2 -19516.125} C_VEL
LIN {X 0,Y 233.28,Z 615.393,A -85,B 0,C 180,E1 -19519.586,E2 -19519.586} C_VEL
LIN {X 0,Y 232.845,Z 617.058,A -85,B 0,C 180,E1 -19523.066,E2 -19523.066} C_VEL
LIN {X 0,Y 232.983,Z 617.424,A -85,B 0,C 180,E1 -19526.541,E2 -19526.541} C_VEL
LIN {X 0,Y 233.227,Z 616.421,A -85,B 0,C 180,E1 -19530,E2 -19530} C_VEL
LIN {X 0,Y 233.091,Z 613.938,A -85,B 0,C 180,E1 -19533.457,E2 -19533.457} C_VEL
LIN {X 0,Y 233.186,Z 611.215,A -85,B 0,C 180,E1 -19535.965,E2 -19535.965} C_VEL
LIN {X 0,Y 233.255,Z 607.278,A -85,B 0,C 180,E1 -19538.664,E2 -19538.664} C_VEL
LIN {X 0,Y 233.855,Z 600.689,A -85,B 0,C 180,E1 -19542.144,E2 -19542.144} C_VEL
LIN {X 0,Y 234.801,Z 593.273,A -85,B 0,C 180,E1 -19545.183,E2 -19545.183} C_VEL
LIN {X 0,Y 236.329,Z 584.359,A -85,B 0,C 180,E1 -19548.105,E2 -19548.105} C_VEL
LIN {X 0,Y 238.159,Z 574.485,A -85,B 0,C 180,E1 -19550.739,E2 -19550.739} C_VEL
LIN {X 0,Y 240.227,Z 563.989,A -85,B 0,C 180,E1 -19553.035,E2 -19553.035} C_VEL
LIN {X 0,Y 242.674,Z 551.349,A -85,B 0,C 180,E1 -19555.288,E2 -19555.288} C_VEL
LIN {X 0,Y 243.114,Z 548.672,A -85,B 0,C 180,E1 -19555.697,E2 -19555.697} C_VEL
LIN {X 0,Y 242.192,Z 537.081,A -85,B 0,C 180,E1 -19557.464,E2 -19557.464} C_VEL
LIN {X 0,Y 240.711,Z 522.578,A -85,B 0,C 180,E1 -19559.333,E2 -19559.333} C_VEL
LIN {X 0,Y 238.813,Z 508.101,A -85,B 0,C 180,E1 -19560.883,E2 -19560.883} C_VEL
LIN {X 0,Y 236.368,Z 492.602,A -85,B 0,C 180,E1 -19562.209,E2 -19562.209} C_VEL
LIN {X 0,Y 235.64,Z 487.998,A -85,B 0,C 180,E1 -19562.559,E2 -19562.559} C_VEL
LIN {X 0,Y 236.715,Z 483.16,A -85,B 0,C 180,E1 -19566.715,E2 -19566.715} C_VEL
LIN {X 0,Y 237.269,Z 479.823,A -85,B 0,C 180,E1 -19569.635,E2 -19569.635} C_VEL
LIN {X 0,Y 237.182,Z 477.009,A -85,B 0,C 180,E1 -19572.202,E2 -19572.202} C_VEL
LIN {X 0,Y 236.58,Z 473.598,A -85,B 0,C 180,E1 -19575.475,E2 -19575.475} C_VEL
LIN {X 0,Y 235.9,Z 470.007,A -85,B 0,C 180,E1 -19579.048,E2 -19579.048} C_VEL
LIN {X 0,Y 235.115,Z 465.126,A -85,B 0,C 180,E1 -19584.199,E2 -19584.199} C_VEL
LIN {X 0,Y 235.026,Z 464.838,A -85,B 0,C 180,E1 -19584.584,E2 -19584.584} C_VEL
LIN {X 0,Y 234.929,Z 464.847,A -85,B 0,C 180,E1 -19589.432,E2 -19589.432} C_VEL
LIN {X 0,Y 234.991,Z 464.833,A -85,B 0,C 180,E1 -19593.794,E2 -19593.794} C_VEL
LIN {X 0,Y 235.008,Z 464.838,A -85,B 0,C 180,E1 -19598.97,E2 -19598.97} C_VEL
LIN {X 0,Y 235.093,Z 464.823,A -85,B 0,C 180,E1 -19603.059,E2 -19603.059} C_VEL
LIN {X 0,Y 235.143,Z 464.817,A -85,B 0,C 180,E1 -19607.924,E2 -19607.924} C_VEL
LIN {X 0,Y 235.373,Z 464.788,A -85,B 0,C 180,E1 -19611.414,E2 -19611.414} C_VEL
LIN {X 0,Y 235.4,Z 464.784,A -85,B 0,C 180,E1 -19613.142,E2 -19613.142} C_VEL
LIN {X 0,Y 235.593,Z 464.763,A -85,B 0,C 180,E1 -19618.291,E2 -19618.291} C_VEL
LIN {X 0,Y 235.595,Z 464.758,A -85,B 0,C 180,E1 -19621.71,E2 -19621.71} C_VEL
LIN {X 0,Y 235.402,Z 464.787,A -85,B 0,C 180,E1 -19626.859,E2 -19626.859} C_VEL
LIN {X 0,Y 235.235,Z 464.807,A -85,B 0,C 180,E1 -19630.327,E2 -19630.327} C_VEL
LIN {X 0,Y 235.109,Z 464.822,A -85,B 0,C 180,E1 -19635.607,E2 -19635.607} C_VEL
LIN {X 0,Y 235.006,Z 464.831,A -85,B 0,C 180,E1 -19639.206,E2 -19639.206} C_VEL
LIN {X 0,Y 234.959,Z 464.841,A -85,B 0,C 180,E1 -19642.883,E2 -19642.883} C_VEL
LIN {X 0,Y 234.968,Z 464.839,A -85,B 0,C 180,E1 -19646.658,E2 -19646.658} C_VEL
LIN {X 0,Y 234.93,Z 464.845,A -85,B 0,C 180,E1 -19650.568,E2 -19650.568} C_VEL
LIN {X 0,Y 234.958,Z 464.84,A -85,B 0,C 180,E1 -19654.634,E2 -19654.634} C_VEL
LIN {X 0,Y 234.941,Z 464.842,A -85,B 0,C 180,E1 -19658.945,E2 -19658.945} C_VEL
LIN {X 0,Y 234.887,Z 464.85,A -85,B 0,C 180,E1 -19663.487,E2 -19663.487} C_VEL
LIN {X 0,Y 234.921,Z 464.844,A -85,B 0,C 180,E1 -19666.523,E2 -19666.523} C_VEL
LIN {X 0,Y 234.955,Z 464.841,A -85,B 0,C 180,E1 -19671.087,E2 -19671.087} C_VEL
LIN {X 0,Y 234.962,Z 464.838,A -85,B 0,C 180,E1 -19675.368,E2 -19675.368} C_VEL
LIN {X 0,Y 234.972,Z 464.84,A -85,B 0,C 180,E1 -19680.158,E2 -19680.158} C_VEL
LIN {X 0,Y 234.997,Z 464.836,A -85,B 0,C 180,E1 -19683.794,E2 -19683.794} C_VEL
LIN {X 0,Y 235.014,Z 464.834,A -85,B 0,C 180,E1 -19688.971,E2 -19688.971} C_VEL
LIN {X 0,Y 235.099,Z 464.821,A -85,B 0,C 180,E1 -19693.06,E2 -19693.06} C_VEL
LIN {X 0,Y 235.118,Z 464.822,A -85,B 0,C 180,E1 -19697.922,E2 -19697.922} C_VEL
LIN {X 0,Y 235.323,Z 464.795,A -85,B 0,C 180,E1 -19701.412,E2 -19701.412} C_VEL
LIN {X 0,Y 235.361,Z 464.791,A -85,B 0,C 180,E1 -19703.14,E2 -19703.14} C_VEL
LIN {X 0,Y 235.599,Z 464.759,A -85,B 0,C 180,E1 -19708.291,E2 -19708.291} C_VEL
LIN {X 0,Y 235.599,Z 464.762,A -85,B 0,C 180,E1 -19711.709,E2 -19711.709} C_VEL
LIN {X 0,Y 235.396,Z 464.787,A -85,B 0,C 180,E1 -19716.859,E2 -19716.859} C_VEL
LIN {X 0,Y 235.218,Z 464.805,A -85,B 0,C 180,E1 -19720.327,E2 -19720.327} C_VEL
LIN {X 0,Y 235.117,Z 464.823,A -85,B 0,C 180,E1 -19725.606,E2 -19725.606} C_VEL
LIN {X 0,Y 235.012,Z 464.837,A -85,B 0,C 180,E1 -19729.205,E2 -19729.205} C_VEL
LIN {X 0,Y 234.964,Z 464.843,A -85,B 0,C 180,E1 -19732.882,E2 -19732.882} C_VEL
LIN {X 0,Y 234.972,Z 464.84,A -85,B 0,C 180,E1 -19736.657,E2 -19736.657} C_VEL
LIN {X 0,Y 234.918,Z 464.848,A -85,B 0,C 180,E1 -19740.569,E2 -19740.569} C_VEL
LIN {X 0,Y 234.841,Z 464.859,A -85,B 0,C 180,E1 -19743.075,E2 -19743.075} C_VEL
LIN {X 0,Y 234.528,Z 464.898,A -85,B 0,C 180,E1 -19746.821,E2 -19746.821} C_VEL
LIN {X 0,Y 234.255,Z 464.933,A -85,B 0,C 180,E1 -19749.747,E2 -19749.747} C_VEL
LIN {X 0,Y 238.725,Z 478.482,A -85,B 0,C 180,E1 -19751.128,E2 -19751.128} C_VEL
LIN {X 0,Y 242.373,Z 492.71,A -85,B 0,C 180,E1 -19752.787,E2 -19752.787} C_VEL
LIN {X 0,Y 245.228,Z 506.055,A -85,B 0,C 180,E1 -19754.597,E2 -19754.597} C_VEL
LIN {X 0,Y 245.862,Z 509.024,A -85,B 0,C 180,E1 -19755.041,E2 -19755.041} C_VEL
LIN {X 0,Y 243.945,Z 521.779,A -85,B 0,C 180,E1 -19756.824,E2 -19756.824} C_VEL
LIN {X 0,Y 241.85,Z 533.355,A -85,B 0,C 180,E1 -19758.798,E2 -19758.798} C_VEL
LIN {X 0,Y 239.91,Z 543.836,A -85,B 0,C 180,E1 -19760.962,E2 -19760.962} C_VEL
LIN {X 0,Y 238.162,Z 553.024,A -85,B 0,C 180,E1 -19763.227,E2 -19763.227} C_VEL
LIN {X 0,Y 236.291,Z 562.788,A -85,B 0,C 180,E1 -19766.158,E2 -19766.158} C_VEL
LIN {X 0,Y 235.009,Z 570.34,A -85,B 0,C 180,E1 -19768.944,E2 -19768.944} C_VEL
LIN {X 0,Y 233.932,Z 577.515,A -85,B 0,C 180,E1 -19772.246,E2 -19772.246} C_VEL
LIN {X 0,Y 233.31,Z 582.328,A -85,B 0,C 180,E1 -19775.056,E2 -19775.056} C_VEL
LIN {X 0,Y 232.895,Z 586.073,A -85,B 0,C 180,E1 -19777.839,E2 -19777.839} C_VEL
LIN {X 0,Y 232.719,Z 588.868,A -85,B 0,C 180,E1 -19780.598,E2 -19780.598} C_VEL
LIN {X 0,Y 232.939,Z 591.168,A -85,B 0,C 180,E1 -19784.244,E2 -19784.244} C_VEL
LIN {X 0,Y 233.538,Z 592.016,A -85,B 0,C 180,E1 -19787.839,E2 -19787.839} C_VEL
LIN {X 0,Y 234.742,Z 591.488,A -85,B 0,C 180,E1 -19791.39,E2 -19791.39} C_VEL
LIN {X 0,Y 236.486,Z 589.631,A -85,B 0,C 180,E1 -19794.885,E2 -19794.885} C_VEL
LIN {X 0,Y 239.041,Z 586.359,A -85,B 0,C 180,E1 -19798.395,E2 -19798.395} C_VEL
LIN {X 0,Y 242.196,Z 581.844,A -85,B 0,C 180,E1 -19801.663,E2 -19801.663} C_VEL
LIN {X 0,Y 246.117,Z 575.762,A -85,B 0,C 180,E1 -19804.914,E2 -19804.914} C_VEL
LIN {X 0,Y 250.216,Z 569.02,A -85,B 0,C 180,E1 -19807.667,E2 -19807.667} C_VEL
LIN {X 0,Y 255.659,Z 559.468,A -85,B 0,C 180,E1 -19810.693,E2 -19810.693} C_VEL
LIN {X 0,Y 260.989,Z 549.173,A -85,B 0,C 180,E1 -19813.261,E2 -19813.261} C_VEL
LIN {X 0,Y 266.474,Z 537.49,A -85,B 0,C 180,E1 -19815.537,E2 -19815.537} C_VEL
LIN {X 0,Y 267.816,Z 534.033,A -85,B 0,C 180,E1 -19816.19,E2 -19816.19} C_VEL
LIN {X 0,Y 267.211,Z 527.396,A -85,B 0,C 180,E1 -19818.398,E2 -19818.398} C_VEL
LIN {X 0,Y 265.981,Z 520.99,A -85,B 0,C 180,E1 -19820.876,E2 -19820.876} C_VEL
LIN {X 0,Y 264.835,Z 517.008,A -85,B 0,C 180,E1 -19822.728,E2 -19822.728} C_VEL
LIN {X 0,Y 263.139,Z 512.674,A -85,B 0,C 180,E1 -19825.298,E2 -19825.298} C_VEL
LIN {X 0,Y 261.654,Z 510.17,A -85,B 0,C 180,E1 -19827.581,E2 -19827.581} C_VEL
LIN {X 0,Y 260.084,Z 507.793,A -85,B 0,C 180,E1 -19830.892,E2 -19830.892} C_VEL
LIN {X 0,Y 259.606,Z 506.994,A -85,B 0,C 180,E1 -19832.943,E2 -19832.943} C_VEL
LIN {X 0,Y 259.245,Z 507.981,A -85,B 0,C 180,E1 -19836.613,E2 -19836.613} C_VEL
LIN {X 0,Y 259.886,Z 509.772,A -85,B 0,C 180,E1 -19839.531,E2 -19839.531} C_VEL
LIN {X 0,Y 261.218,Z 515.269,A -85,B 0,C 180,E1 -19843.413,E2 -19843.413} C_VEL
LIN {X 0,Y 261.605,Z 516.616,A -85,B 0,C 180,E1 -19844.159,E2 -19844.159} C_VEL
LIN {X 0,Y 261.841,Z 518.392,A -85,B 0,C 180,E1 -19844.922,E2 -19844.922} C_VEL
LIN {X 0,Y 261.594,Z 521.969,A -85,B 0,C 180,E1 -19845.954,E2 -19845.954} C_VEL
LIN {X 0,Y 260.828,Z 526.137,A -85,B 0,C 180,E1 -19846.877,E2 -19846.877} C_VEL
LIN {X 0,Y 258.955,Z 534.903,A -85,B 0,C 180,E1 -19848.721,E2 -19848.721} C_VEL
LIN {X 0,Y 258.66,Z 537.501,A -85,B 0,C 180,E1 -19849.412,E2 -19849.412} C_VEL
LIN {X 0,Y 257.827,Z 547.01,A -85,B 0,C 180,E1 -19852.01,E2 -19852.01} C_VEL
LIN {X 0,Y 256.051,Z 556.555,A -85,B 0,C 180,E1 -19854.391,E2 -19854.391} C_VEL
LIN {X 0,Y 253.736,Z 564.204,A -85,B 0,C 180,E1 -19856.195,E2 -19856.195} C_VEL
LIN {X 0,Y 247.657,Z 575.914,A -85,B 0,C 180,E1 -19858.809,E2 -19858.809} C_VEL
LIN {X 0,Y 242.515,Z 585.253,A -85,B 0,C 180,E1 -19861.435,E2 -19861.435} C_VEL
LIN {X 0,Y 238.107,Z 593.092,A -85,B 0,C 180,E1 -19864.192,E2 -19864.192} C_VEL
LIN {X 0,Y 234.363,Z 599.695,A -85,B 0,C 180,E1 -19867.056,E2 -19867.056} C_VEL
LIN {X 0,Y 230.928,Z 605.774,A -85,B 0,C 180,E1 -19870.442,E2 -19870.442} C_VEL
LIN {X 0,Y 228.436,Z 610.498,A -85,B 0,C 180,E1 -19873.926,E2 -19873.926} C_VEL
LIN {X 0,Y 226.741,Z 613.899,A -85,B 0,C 180,E1 -19877.469,E2 -19877.469} C_VEL
LIN {X 0,Y 225.925,Z 616.047,A -85,B 0,C 180,E1 -19881.052,E2 -19881.052} C_VEL
LIN {X 0,Y 225.807,Z 616.928,A -85,B 0,C 180,E1 -19884.85,E2 -19884.85} C_VEL
LIN {X 0,Y 225.915,Z 616.872,A -85,B 0,C 180,E1 -19886.433,E2 -19886.433} C_VEL
LIN {X 0,Y 226.153,Z 615.732,A -85,B 0,C 180,E1 -19890,E2 -19890} C_VEL
LIN {X 0,Y 226.033,Z 613.104,A -85,B 0,C 180,E1 -19893.565,E2 -19893.565} C_VEL
LIN {X 0,Y 226.117,Z 610.526,A -85,B 0,C 180,E1 -19895.958,E2 -19895.958} C_VEL
LIN {X 0,Y 226.205,Z 606.223,A -85,B 0,C 180,E1 -19898.937,E2 -19898.937} C_VEL
LIN {X 0,Y 226.645,Z 601.301,A -85,B 0,C 180,E1 -19901.628,E2 -19901.628} C_VEL
LIN {X 0,Y 227.547,Z 594.188,A -85,B 0,C 180,E1 -19904.762,E2 -19904.762} C_VEL
LIN {X 0,Y 228.841,Z 586.205,A -85,B 0,C 180,E1 -19907.599,E2 -19907.599} C_VEL
LIN {X 0,Y 230.457,Z 577.776,A -85,B 0,C 180,E1 -19910.064,E2 -19910.064} C_VEL
LIN {X 0,Y 232.522,Z 567.021,A -85,B 0,C 180,E1 -19912.666,E2 -19912.666} C_VEL
LIN {X 0,Y 234.703,Z 556.288,A -85,B 0,C 180,E1 -19914.785,E2 -19914.785} C_VEL
LIN {X 0,Y 236.123,Z 548.768,A -85,B 0,C 180,E1 -19916.041,E2 -19916.041} C_VEL
LIN {X 0,Y 235.045,Z 535.721,A -85,B 0,C 180,E1 -19918.094,E2 -19918.094} C_VEL
LIN {X 0,Y 233.691,Z 521.895,A -85,B 0,C 180,E1 -19919.923,E2 -19919.923} C_VEL
LIN {X 0,Y 231.797,Z 507.723,A -85,B 0,C 180,E1 -19921.489,E2 -19921.489} C_VEL
LIN {X 0,Y 229.427,Z 492.301,A -85,B 0,C 180,E1 -19922.842,E2 -19922.842} C_VEL
LIN {X 0,Y 228.701,Z 487.629,A -85,B 0,C 180,E1 -19923.213,E2 -19923.213} C_VEL
LIN {X 0,Y 229.868,Z 482.593,A -85,B 0,C 180,E1 -19927.696,E2 -19927.696} C_VEL
LIN {X 0,Y 230.227,Z 479.794,A -85,B 0,C 180,E1 -19930.257,E2 -19930.257} C_VEL
LIN {X 0,Y 230.008,Z 477.085,A -85,B 0,C 180,E1 -19932.834,E2 -19932.834} C_VEL
LIN {X 0,Y 229.375,Z 473.48,A -85,B 0,C 180,E1 -19936.408,E2 -19936.408} C_VEL
LIN {X 0,Y 228.643,Z 469.845,A -85,B 0,C 180,E1 -19940.214,E2 -19940.214} C_VEL
LIN {X 0,Y 227.962,Z 465.717,A -85,B 0,C 180,E1 -19944.822,E2 -19944.822} C_VEL
LIN {X 0,Y 227.916,Z 465.72,A -85,B 0,C 180,E1 -19950.438,E2 -19950.438} C_VEL
LIN {X 0,Y 227.926,Z 465.714,A -85,B 0,C 180,E1 -19954.426,E2 -19954.426} C_VEL
LIN {X 0,Y 227.959,Z 465.712,A -85,B 0,C 180,E1 -19958.287,E2 -19958.287} C_VEL
LIN {X 0,Y 228.031,Z 465.705,A -85,B 0,C 180,E1 -19962.826,E2 -19962.826} C_VEL
LIN {X 0,Y 228.09,Z 465.696,A -85,B 0,C 180,E1 -19967.545,E2 -19967.545} C_VEL
LIN {X 0,Y 228.303,Z 465.669,A -85,B 0,C 180,E1 -19971.146,E2 -19971.146} C_VEL
LIN {X 0,Y 228.351,Z 465.663,A -85,B 0,C 180,E1 -19972.929,E2 -19972.929} C_VEL
LIN {X 0,Y 228.552,Z 465.64,A -85,B 0,C 180,E1 -19978.238,E2 -19978.238} C_VEL
LIN {X 0,Y 228.554,Z 465.635,A -85,B 0,C 180,E1 -19981.762,E2 -19981.762} C_VEL
LIN {X 0,Y 228.353,Z 465.664,A -85,B 0,C 180,E1 -19987.072,E2 -19987.072} C_VEL
LIN {X 0,Y 228.16,Z 465.687,A -85,B 0,C 180,E1 -19990.651,E2 -19990.651} C_VEL
LIN {X 0,Y 228.06,Z 465.703,A -85,B 0,C 180,E1 -19994.273,E2 -19994.273} C_VEL
LIN {X 0,Y 228.001,Z 465.708,A -85,B 0,C 180,E1 -19997.954,E2 -19997.954} C_VEL
LIN {X 0,Y 227.928,Z 465.719,A -85,B 0,C 180,E1 -20002.33,E2 -20002.33} C_VEL
LIN {X 0,Y 227.941,Z 465.714,A -85,B 0,C 180,E1 -20006.604,E2 -20006.604} C_VEL
LIN {X 0,Y 227.907,Z 465.722,A -85,B 0,C 180,E1 -20010.297,E2 -20010.297} C_VEL
LIN {X 0,Y 227.887,Z 465.723,A -85,B 0,C 180,E1 -20013.719,E2 -20013.719} C_VEL
LIN {X 0,Y 227.847,Z 465.727,A -85,B 0,C 180,E1 -20018.091,E2 -20018.091} C_VEL
LIN {X 0,Y 227.811,Z 465.731,A -85,B 0,C 180,E1 -20022.743,E2 -20022.743} C_VEL
LIN {X 0,Y 227.864,Z 465.723,A -85,B 0,C 180,E1 -20027.271,E2 -20027.271} C_VEL
LIN {X 0,Y 227.872,Z 465.726,A -85,B 0,C 180,E1 -20031.915,E2 -20031.915} C_VEL
LIN {X 0,Y 227.892,Z 465.721,A -85,B 0,C 180,E1 -20036.374,E2 -20036.374} C_VEL
LIN {X 0,Y 227.922,Z 465.717,A -85,B 0,C 180,E1 -20040.439,E2 -20040.439} C_VEL
LIN {X 0,Y 227.931,Z 465.714,A -85,B 0,C 180,E1 -20044.427,E2 -20044.427} C_VEL
LIN {X 0,Y 227.965,Z 465.712,A -85,B 0,C 180,E1 -20048.288,E2 -20048.288} C_VEL
LIN {X 0,Y 228.038,Z 465.7,A -85,B 0,C 180,E1 -20052.826,E2 -20052.826} C_VEL
LIN {X 0,Y 228.076,Z 465.702,A -85,B 0,C 180,E1 -20057.544,E2 -20057.544} C_VEL
LIN {X 0,Y 228.261,Z 465.674,A -85,B 0,C 180,E1 -20061.144,E2 -20061.144} C_VEL
LIN {X 0,Y 228.313,Z 465.667,A -85,B 0,C 180,E1 -20062.927,E2 -20062.927} C_VEL
LIN {X 0,Y 228.557,Z 465.636,A -85,B 0,C 180,E1 -20068.238,E2 -20068.238} C_VEL
LIN {X 0,Y 228.558,Z 465.639,A -85,B 0,C 180,E1 -20071.762,E2 -20071.762} C_VEL
LIN {X 0,Y 228.343,Z 465.666,A -85,B 0,C 180,E1 -20077.072,E2 -20077.072} C_VEL
LIN {X 0,Y 228.149,Z 465.686,A -85,B 0,C 180,E1 -20080.651,E2 -20080.651} C_VEL
LIN {X 0,Y 228.068,Z 465.7,A -85,B 0,C 180,E1 -20084.272,E2 -20084.272} C_VEL
LIN {X 0,Y 228.006,Z 465.705,A -85,B 0,C 180,E1 -20087.953,E2 -20087.953} C_VEL
